# B&R Automation Studio project NAEUL004C00R13L518F00 (part 39)

#### Act_Main.st - Do Not Change!!!
```iecst
(** 2019-07-03 **)
ACTION Act_Main:

	fbMagPresentTm(IN := tylocalBuffer.In.bMagPresentSensor);

	//Update Retain
	IF bUpdateSensor = TRUE THEN
		tylocalBuffer.Out.bMagPresent	:= fbMagPresentTm.Q;
	END_IF

	//Display Buffer
	IF bUpdtDisplay = TRUE THEN
		fDispBffrDescending(ADR(tylocalBuffer.In.tyDispBuffer) , tyBffrParameter , tylocalBuffer.In.tyBuffer , tylocalBuffer.In.dtCurrDT , DINT_TO_TIME(tylocalBuffer.In.diCoolTm) , 0 , 1 , 2);
	END_IF

	//Cooling Fan Control
	IF tylocalBuffer.In.bManual = TRUE THEN
		;

	ELSIF bCoolFanRun = TRUE AND tylocalBuffer.In.bPrepCoolFan = TRUE AND bCoolFanTm = TRUE THEN //Cooling Fan Control By Cooling Time

		fbCoolFanOffChkTm(IN := TRUE);

		IF fbCoolFanOffChkTm.Q = TRUE THEN
			IF fBffrChkCoolBrdAny(tylocalBuffer.In.dtCurrDT, DINT_TO_TIME(tylocalBuffer.In.diCoolTm), tylocalBuffer.In.tyBuffer) = 0 THEN
				fbCoolFanOffDlyTm.IN	:= TRUE;
			ELSE
				fbCoolFanOffDlyTm.IN	:= FALSE;
				tylocalBuffer.Out.bCoolFanCtrl			:= TRUE;
			END_IF

			fbCoolFanOffChkTm(IN := FALSE);
		END_IF

		fbCoolFanOffDlyTm;

		IF fbCoolFanOffDlyTm.Q = TRUE THEN
			tylocalBuffer.Out.bCoolFanCtrl	:= FALSE;
		END_IF

	ELSIF bCoolFanRun = TRUE AND tylocalBuffer.In.bPrepCoolFan = TRUE AND bCoolFanTm = FALSE THEN	//Cooling Fan Control By Buffer Empty
		fbCoolFanOffDlyTm(IN := tylocalBuffer.In.tyBufferStat.bBffrMty);

		IF tylocalBuffer.In.tyBufferStat.bBffrMty = FALSE THEN
			tylocalBuffer.Out.bCoolFanCtrl	:= TRUE;
		END_IF

		IF fbCoolFanOffDlyTm.Q = TRUE THEN
			tylocalBuffer.Out.bCoolFanCtrl	:= FALSE;
		END_IF

	ELSE

		tylocalBuffer.Out.bCoolFanCtrl	:= FALSE;

	END_IF

	//Set Buffer By Magazine Present
	IF bBffrSetFull = TRUE THEN
		IF tylocalBuffer.In.bMagPresentSensor = TRUE AND fbMagAbsentTm.Q = TRUE THEN
			bSetFull		:= TRUE;
			tylocalBuffer.Out.dtMagPresentTm	:= tylocalBuffer.In.dtCurrDT;
		END_IF

		IF bSetFull = TRUE  THEN
			tylocalBuffer.In.eAct	:= BufferActSetFull;

			IF eStatus = Done AND eStat = BufferActSetFull THEN
				tylocalBuffer.In.eAct		:= BufferActIdle;
				bSetFull	:= FALSE;
			ELSIF eStatus = Error THEN
				bSetFull	:= FALSE;
			END_IF
		END_IF

		fbMagAbsentTm(IN := NOT tylocalBuffer.In.bMagPresentSensor);

	ELSIF bBffrSetMty = TRUE THEN
		IF tylocalBuffer.In.bMagPresentSensor = TRUE AND fbMagAbsentTm.Q = TRUE THEN
			bSetMty			:= TRUE;
			tylocalBuffer.Out.dtMagPresentTm	:= tylocalBuffer.In.dtCurrDT;
		END_IF

		IF bSetMty = TRUE  THEN
			tylocalBuffer.In.eAct	:= BufferActSetMty;

			IF eStatus = Done AND eStat = BufferActSetMty THEN
				tylocalBuffer.In.eAct	:= BufferActIdle;
				bSetMty	:= FALSE;
			ELSIF eStatus = Error THEN
				bSetMty	:= FALSE;
			END_IF
		END_IF

		fbMagAbsentTm(IN := NOT tylocalBuffer.In.bMagPresentSensor);

	END_IF
	//background--end//

	//Check Parameter Different
	tylocalBuffer.Out.bParamDiff	:= (tyBffrParameter.bAscending <> tylocalBuffer.In.bAscending)
	OR (tyBffrParameter.diMinSlt <> tylocalBuffer.In.diMinSlt)
	OR (tyBffrParameter.diMaxSlt <> tylocalBuffer.In.diMaxSlt)
	OR (tyBffrParameter.diPitch <> tylocalBuffer.In.diPitch)
	OR (tyBffrParameter.diSltCap <> tylocalBuffer.In.diSltCap)
	OR (tylocalBuffer.Out.bFIFOOld <> tylocalBuffer.In.bFIFO);

	//Update MagRemoved
	tylocalBuffer.Out.bMagRemoved	:= fbMagAbsentTm.Q;

	//Action
	IF tylocalBuffer.Out.eStatus = Idle OR tylocalBuffer.Out.eStatus = Busy OR tylocalBuffer.Out.eStatus = Done THEN
		tylocalBuffer.Out.eStat	:= tylocalBuffer.In.eAct;
	END_IF

	IF eStatOld <> tylocalBuffer.Out.eStat THEN
		fbDirCreate1(bEn := FALSE);
		fbDirCreate2(bEn := FALSE);
		fbFileRead1(bEn := FALSE);
		fbFileWrite1(bEn := FALSE);
		usiStep	:= 0;

		bFileNotFound			:= FALSE;
		bNewProduct				:= FALSE;
		bLastProductUnload		:= FALSE;
		bLastProductLeftInBffr	:= FALSE;

		tylocalBuffer.Out.sStatTxt	:= a_sStatText[tylocalBuffer.Out.eStat];

		eStatOld	:= tylocalBuffer.Out.eStat;

		tylocalBuffer.Out.eStatus		:= Busy;
	END_IF

	//Main
	CASE tylocalBuffer.Out.eStat OF

		BufferActIdle:
			tylocalBuffer.Out.eStatus	:= Idle;

		BufferActCreateDir:
			IF tylocalBuffer.Out.eStatus = Idle OR tylocalBuffer.Out.eStatus = Busy THEN

				tylocalBuffer.Out.eStatus	:= Busy;

				CASE usiStep OF
					0:
						fbDirCreate1(bEn := TRUE);
						IF fbDirCreate1.udiStatus = 0 THEN
							usiStep	:= 1;
						ELSIF fbDirCreate1.udiStatus < 65534 THEN
							tylocalBuffer.Out.eStatus		:= Error;

							IF fbDirCreate1.udiStatus = 1908 THEN
								udiStatus	:= 10000;	//Create User Directory Error
							ELSE
								udiStatus	:= fbDirCreate1.udiStatus;
							END_IF
						END_IF

					1:
						fbDirCreate2(bEn := TRUE);
						IF fbDirCreate2.udiStatus = 0 THEN
							tylocalBuffer.Out.eStatus	:= Done;
						ELSIF fbDirCreate2.udiStatus < 65534 THEN
							tylocalBuffer.Out.eStatus		:= Error;

							IF fbDirCreate2.udiStatus = 1908 THEN
								udiStatus	:= 10001;	//Create Retain Directory Error
							ELSE
								udiStatus	:= fbDirCreate2.udiStatus;
							END_IF
						END_IF

				END_CASE

			END_IF

		BufferActGetRetainBffr:
			IF tylocalBuffer.Out.eStatus = Idle OR tylocalBuffer.Out.eStatus = Busy THEN

				tylocalBuffer.Out.eStatus	:= Busy;

				fbFileRead1(bEn := TRUE);
				IF fbFileRead1.udiStatus = 0 THEN
					tylocalBuffer.Out.eStatus	:= Done;

					tyBffrParameter.diBffrTtlSlt	:= tylocalBuffer.In.diBffrTtlSlt;
					tyBffrParameter.diSltCap		:= tylocalBuffer.In.diSltCap;

					fBffrStat(ADR(tylocalBuffer.In.tylocalBuffer.Out.tylocalBuffer.Out.tyBufferStat) , tylocalBuffer.In.tylocalBuffer.Out.tyBuffer);
					fDispBffrDescending(ADR(tylocalBuffer.In.tylocalBuffer.Out.tyDispBuffer) , tyBffrParameter , tylocalBuffer.In.tylocalBuffer.Out.tyBuffer , tylocalBuffer.In.dtCurrDT , DINT_TO_TIME(tylocalBuffer.In.diCoolTm) , 0 , 1 , 2);

				ELSIF fbFileRead1.udiStatus < 65534 THEN
					tylocalBuffer.Out.eStatus	:= Error;

					IF fbFileRead1.udiStatus = 1900 THEN
						udiStatus	:= 10002;	//File Open Error While Reading Retain File
					ELSIF fbFileRead1.udiStatus = 1902 THEN
						udiStatus	:= 10003;	//File Read Error While Reading Retain File
					ELSIF fbFileRead1.udiStatus = 1904 THEN
						udiStatus	:= 10004;	//File Close Error While Reading Retain File
					ELSIF fbFileRead1.udiStatus = 1915 THEN
						tylocalBuffer.Out.eStatus			:= Done;
						bFileNotFound	:= TRUE;
					ELSE
						udiStatus	:= fbFileRead1.udiStatus;
					END_IF
				END_IF

			END_IF

		BufferActSetFull:
			IF tylocalBuffer.Out.eStatus = Idle OR tylocalBuffer.Out.eStatus = Busy THEN

				tylocalBuffer.Out.eStatus	:= Busy;

				CASE usiStep OF
					0:
						tyBffrParameter.bAscending		:= tylocalBuffer.In.bAscending;
						tyBffrParameter.diBffrTtlSlt	:= tylocalBuffer.In.diBffrTtlSlt;
						tyBffrParameter.diMaxSlt		:= tylocalBuffer.In.diMaxSlt;
						tyBffrParameter.diMinSlt		:= tylocalBuffer.In.diMinSlt;
						tyBffrParameter.diPitch			:= tylocalBuffer.In.diPitch;
						tyBffrParameter.diSltCap		:= tylocalBuffer.In.diSltCap;
						tyBffrParameter.a_bSkip			:= tylocalBuffer.In.a_bSkip;
						tylocalBuffer.Out.bFIFOOld		:= tylocalBuffer.In.bFIFO;

						udiStatus	:= fBffrSetFull(ADR(tylocalBuffer.In.tylocalBuffer.Out.tyBuffer) , tyBffrParameter , tylocalBuffer.In.dtCurrDT , tylocalBuffer.In.sBffrNm , tylocalBuffer.In.sProdNm);

						IF udiStatus = 0 THEN
							usiStep	:= 1;

							fBffrStat(ADR(tylocalBuffer.In.tylocalBuffer.Out.tylocalBuffer.Out.tyBufferStat) , tylocalBuffer.In.tylocalBuffer.Out.tyBuffer);
							fDispBffrDescending(ADR(tylocalBuffer.In.tylocalBuffer.Out.tyDispBuffer) , tyBffrParameter , tylocalBuffer.In.tylocalBuffer.Out.tyBuffer , tylocalBuffer.In.dtCurrDT , DINT_TO_TIME(tylocalBuffer.In.diCoolTm) , 0 , 1 , 2);

						ELSE
							tylocalBuffer.Out.eStatus	:= Error;

						END_IF

					1:
						fbFileWrite1(bEn := TRUE);

						IF fbFileWrite1.udiStatus = 0 THEN
							tylocalBuffer.Out.eStatus	:= Done;
						ELSIF fbFileWrite1.udiStatus < 65534 THEN
							tylocalBuffer.Out.eStatus	:= Error;

							IF fbFileWrite1.udiStatus = 1900 THEN
								udiStatus	:= 10005;	//File Open Error While Setting Full Buffer
							ELSIF fbFileWrite1.udiStatus = 1901 THEN
								udiStatus	:= 10006;	//File Create Error While Setting Full Buffer
							ELSIF fbFileWrite1.udiStatus = 1903 THEN
								udiStatus	:= 10007;	//File Write Error While Setting Full Buffer
							ELSIF fbFileWrite1.udiStatus = 1904 THEN
								udiStatus	:= 10008;	//File Close Error While Setting Full Buffer
							ELSIF fbFileWrite1.udiStatus = 1914 THEN
								udiStatus	:= 10040;	//Directory Does Not Exist While Setting Full Buffer
							ELSE
								udiStatus	:= fbFileWrite1.udiStatus;
							END_IF
						END_IF

				END_CASE

			END_IF

		BufferActSetMty:
			IF tylocalBuffer.Out.eStatus = Idle OR tylocalBuffer.Out.eStatus = Busy THEN

				tylocalBuffer.Out.eStatus	:= Busy;

				CASE usiStep OF
					0:
						tyBffrParameter.bAscending		:= tylocalBuffer.In.bAscending;
						tyBffrParameter.diBffrTtlSlt	:= tylocalBuffer.In.diBffrTtlSlt;
						tyBffrParameter.diMaxSlt		:= tylocalBuffer.In.diMaxSlt;
						tyBffrParameter.diMinSlt		:= tylocalBuffer.In.diMinSlt;
						tyBffrParameter.diPitch			:= tylocalBuffer.In.diPitch;
						tyBffrParameter.diSltCap		:= tylocalBuffer.In.diSltCap;
						tyBffrParameter.a_bSkip			:= tylocalBuffer.In.a_bSkip;
						tylocalBuffer.Out.bFIFOOld						:= tylocalBuffer.In.bFIFO;

						udiStatus	:= fBffrSetMty(ADR(tylocalBuffer.In.tylocalBuffer.Out.tyBuffer) , tyBffrParameter , tylocalBuffer.In.sBffrNm);

						IF udiStatus = 0 THEN
							usiStep	:= 1;

							fBffrStat(ADR(tylocalBuffer.In.tylocalBuffer.Out.tylocalBuffer.Out.tyBufferStat) , tylocalBuffer.In.tylocalBuffer.Out.tyBuffer);
							fDispBffrDescending(ADR(tylocalBuffer.In.tylocalBuffer.Out.tyDispBuffer) , tyBffrParameter , tylocalBuffer.In.tylocalBuffer.Out.tyBuffer , tylocalBuffer.In.dtCurrDT , DINT_TO_TIME(tylocalBuffer.In.diCoolTm) , 0 , 1 , 2);

						ELSE
							tylocalBuffer.Out.eStatus	:= Error;

						END_IF

					1:
						fbFileWrite1(bEn := TRUE);

						IF fbFileWrite1.udiStatus = 0 THEN
							tylocalBuffer.Out.eStatus	:= Done;
						ELSIF fbFileWrite1.udiStatus < 65534 THEN
							tylocalBuffer.Out.eStatus	:= Error;

							IF fbFileWrite1.udiStatus = 1900 THEN
								udiStatus	:= 10009;	//File Open Error While Setting Empty Buffer
							ELSIF fbFileWrite1.udiStatus = 1901 THEN
								udiStatus	:= 10010;	//File Create Error While Setting Empty Buffer
							ELSIF fbFileWrite1.udiStatus = 1903 THEN
								udiStatus	:= 10011;	//File Write Error While Setting Empty Buffer
							ELSIF fbFileWrite1.udiStatus = 1904 THEN
								udiStatus	:= 10012;	//File Close Error While Setting Empty Buffer
							ELSIF fbFileWrite1.udiStatus = 1914 THEN
								udiStatus	:= 10041;	//Directory Does Not Exist While Setting Empty Buffer
							ELSE
								udiStatus	:= fbFileWrite1.udiStatus;
							END_IF
						END_IF

				END_CASE

			END_IF

		BufferActLoad:
			IF tylocalBuffer.Out.eStatus = Idle OR tylocalBuffer.Out.eStatus = Busy THEN

				tylocalBuffer.Out.eStatus	:= Busy;

				CASE usiStep OF
					0:
						tyLocalBuffer.Out.diCurrSlt	:= fLifterPosInUMToSltBtmMin(tylocalBuffer.In.diLifterCurrPosInUM , tylocalBuffer.In.diSltToSltInUM , tylocalBuffer.In.diLifterBtmPosInUM);

						udiStatus	:= fBffrLoad(ADR(tylocalBuffer.In.tylocalBuffer.Out.tyBuffer) , ADR(bNewProduct) , tyLocalBuffer.Out.diCurrSlt , tylocalBuffer.In.dtCurrDT , tylocalBuffer.In.bGdBrdIn , tylocalBuffer.In.sProdNm , tylocalBuffer.In.sBarcode1 , tylocalBuffer.In.sBarcode2);

						IF udiStatus = 0 THEN
							usiStep	:= 1;

							tyBffrParameter.diBffrTtlSlt	:= tylocalBuffer.In.diBffrTtlSlt;
							tyBffrParameter.diSltCap		:= tylocalBuffer.In.diSltCap;

							fBffrStat(ADR(tylocalBuffer.In.tylocalBuffer.Out.tylocalBuffer.Out.tyBufferStat) , tylocalBuffer.In.tylocalBuffer.Out.tyBuffer);
							fDispBffrDescending(ADR(tylocalBuffer.In.tylocalBuffer.Out.tyDispBuffer) , tyBffrParameter , tylocalBuffer.In.tylocalBuffer.Out.tyBuffer , tylocalBuffer.In.dtCurrDT , DINT_TO_TIME(tylocalBuffer.In.diCoolTm) , 0 , 1 , 2);

						ELSE
							tylocalBuffer.Out.eStatus	:= Error;

							IF udiStatus = 1010 THEN
								udiStatus	:= 10076;	//Loading Slot Is Not For Board
							ELSIF udiStatus = 1011 THEN
								udiStatus	:= 10077;	//Loading Slot Is Full Of Board
							ELSIF udiStatus = 1012 THEN
								udiStatus	:= 10078;	//Loading First Sub-Slot Is Not For Board
							ELSIF udiStatus	= 1013 THEN
								udiStatus	:= 10079;	//Loading Last Sub-Slot Have Board, Which Mean Slot Is Full Of Board
							ELSIF udiStatus = 1014 THEN
								udiStatus	:= 10080;	//Loading Last Sub-Slot Is Not For Board
							ELSIF udiStatus = 1015 THEN
								udiStatus	:= 10081;	//Loading Slot Is Full Of Board
							ELSIF udiStatus = 1001 THEN
								udiStatus	:= 10082;	//Loading Slot Is Skipped
							ELSIF udiStatus	= 1016 THEN
								udiStatus	:= 10083;	//Existing Board Status Is Different With Loading Board Status
							END_IF

						END_IF

					1:
						fbFileWrite1(bEn := TRUE);

						IF fbFileWrite1.udiStatus = 0 THEN
							tylocalBuffer.Out.eStatus	:= Done;
						ELSIF fbFileWrite1.udiStatus < 65534 THEN
							tylocalBuffer.Out.eStatus	:= Error;

							IF fbFileWrite1.udiStatus = 1900 THEN
								udiStatus	:= 10013;	//File Open Error While Loading Info To Buffer
							ELSIF fbFileWrite1.udiStatus = 1901 THEN
								udiStatus	:= 10014;	//File Create Error While Loading Info To Buffer
							ELSIF fbFileWrite1.udiStatus = 1903 THEN
								udiStatus	:= 10015;	//File Write Error While Loading Info To Buffer
							ELSIF fbFileWrite1.udiStatus = 1904 THEN
								udiStatus	:= 10016;	//File Close Error While Loading Info To Buffer
							ELSIF fbFileWrite1.udiStatus = 1914 THEN
								udiStatus	:= 10042;	//Directory Does Not Exist While Loading Info To Buffer
							ELSE
								udiStatus	:= fbFileWrite1.udiStatus;
							END_IF
						END_IF

				END_CASE

			END_IF

		BufferActLoadSltChk:
			IF tylocalBuffer.Out.eStatus = Idle OR tylocalBuffer.Out.eStatus = Busy THEN

				tylocalBuffer.Out.eStatus	:= Busy;

				CASE usiStep OF
					0:
						tyLocalBuffer.Out.diCurrSlt	:= fLifterPosInUMToSltBtmMin(tylocalBuffer.In.diLifterCurrPosInUM , tylocalBuffer.In.diSltToSltInUM , tylocalBuffer.In.diLifterBtmPosInUM);

						IF tylocalBuffer.In.bNxtLoadSeq = TRUE AND tylocalBuffer.In.bGdBrdIn = TRUE THEN
							diExpectedSlt	:= fBffrNxtLoadSeqGd(tylocalBuffer.In.bAscending , tylocalBuffer.In.tylocalBuffer.Out.tyBuffer);
						ELSIF tylocalBuffer.In.bNxtLoadSeq = TRUE AND tylocalBuffer.In.bGdBrdIn = FALSE THEN
							diExpectedSlt	:= fBffrNxtLoadSeqBad(tylocalBuffer.In.bAscending , tylocalBuffer.In.tylocalBuffer.Out.tyBuffer);
						ELSIF tylocalBuffer.In.bNxtLoadSeq = FALSE AND tylocalBuffer.In.bGdBrdIn = TRUE THEN
							diExpectedSlt	:= fBffrNxtLoadNearbyGd(tyLocalBuffer.Out.diCurrSlt , tylocalBuffer.In.tylocalBuffer.Out.tyBuffer);
						ELSE
							diExpectedSlt	:= fBffrNxtLoadNearbyBad(tyLocalBuffer.Out.diCurrSlt , tylocalBuffer.In.tylocalBuffer.Out.tyBuffer);
						END_IF

						IF tyLocalBuffer.Out.diCurrSlt = diExpectedSlt THEN
							udiStatus	:= fBffrLoad(ADR(tylocalBuffer.In.tylocalBuffer.Out.tyBuffer) , ADR(bNewProduct) , tyLocalBuffer.Out.diCurrSlt , tylocalBuffer.In.dtCurrDT , tylocalBuffer.In.bGdBrdIn , tylocalBuffer.In.sProdNm , tylocalBuffer.In.sBarcode1 , tylocalBuffer.In.sBarcode2);

							IF udiStatus = 0 THEN
								usiStep	:= 1;

								tyBffrParameter.diBffrTtlSlt	:= tylocalBuffer.In.diBffrTtlSlt;
								tyBffrParameter.diSltCap		:= tylocalBuffer.In.diSltCap;

								fBffrStat(ADR(tylocalBuffer.In.tylocalBuffer.Out.tylocalBuffer.Out.tyBufferStat) , tylocalBuffer.In.tylocalBuffer.Out.tyBuffer);
								fDispBffrDescending(ADR(tylocalBuffer.In.tylocalBuffer.Out.tyDispBuffer) , tyBffrParameter , tylocalBuffer.In.tylocalBuffer.Out.tyBuffer , tylocalBuffer.In.dtCurrDT , DINT_TO_TIME(tylocalBuffer.In.diCoolTm) , 0 , 1 , 2);

							ELSE
								tylocalBuffer.Out.eStatus	:= Error;

								IF udiStatus = 1010 THEN
									udiStatus	:= 10084;	//Loading Slot Is Not For Board
								ELSIF udiStatus = 1011 THEN
									udiStatus	:= 10085;	//Loading Slot Is Full Of Board
								ELSIF udiStatus = 1012 THEN
									udiStatus	:= 10086;	//Loading First Sub-Slot Is Not For Board
								ELSIF udiStatus	= 1013 THEN
									udiStatus	:= 10087;	//Loading Last Sub-Slot Have Board, Which Mean Slot Is Full Of Board
								ELSIF udiStatus = 1014 THEN
									udiStatus	:= 10088;	//Loading Last Sub-Slot Is Not For Board
								ELSIF udiStatus = 1015 THEN
									udiStatus	:= 10089;	//Loading Slot Is Full Of Board
								ELSIF udiStatus = 1001 THEN
									udiStatus	:= 10090;	//Loading Slot Is Skipped
								ELSIF udiStatus	= 1016 THEN
									udiStatus	:= 10091;	//Existing Board Status Is Different With Loading Board Status
								END_IF

							END_IF

						ELSE
							udiStatus	:= 10017;	//Wrong Slot Number To Load
							tylocalBuffer.Out.eStatus		:= Error;

						END_IF

					1:
						fbFileWrite1(bEn := TRUE);

						IF fbFileWrite1.udiStatus = 0 THEN
							tylocalBuffer.Out.eStatus	:= Done;
						ELSIF fbFileWrite1.udiStatus < 65534 THEN
							tylocalBuffer.Out.eStatus	:= Error;

							IF fbFileWrite1.udiStatus = 1900 THEN
								udiStatus	:= 10018;	//File Open Error While Loading Info To Buffer With Slot Check
							ELSIF fbFileWrite1.udiStatus = 1901 THEN
								udiStatus	:= 10019;	//File Create Error While Loading Info To Buffer With Slot Check
							ELSIF fbFileWrite1.udiStatus = 1903 THEN
								udiStatus	:= 10020;	//File Write Error While Loading Info To Buffer With Slot Check
							ELSIF fbFileWrite1.udiStatus = 1904 THEN
								udiStatus	:= 10021;	//File Close Error While Loading Info To Buffer With Slot Check
							ELSIF fbFileWrite1.udiStatus = 1914 THEN
								udiStatus	:= 10043;	//Directory Does Not Exist While Loading Info To Buffer With Slot Check
							ELSE
								udiStatus	:= fbFileWrite1.udiStatus;
							END_IF
						END_IF

				END_CASE

			END_IF

		BufferActUnload:
			IF tylocalBuffer.Out.eStatus = Idle OR tylocalBuffer.Out.eStatus = Busy THEN

				tylocalBuffer.Out.eStatus	:= Busy;

				CASE usiStep OF
					0:
						tyLocalBuffer.Out.diCurrSlt	:= fLifterPosInUMToSltBtmMin(tylocalBuffer.In.diLifterCurrPosInUM , tylocalBuffer.In.diSltToSltInUM , tylocalBuffer.In.diLifterBtmPosInUM);

						udiStatus	:= fBffrUnload(ADR(tylocalBuffer.Out.tyBoardUnloadStat) , ADR(tylocalBuffer.In.tylocalBuffer.Out.tyBuffer) , ADR(bLastProductUnload) , ADR(bLastProductLeftInBffr) , tyLocalBuffer.Out.diCurrSlt);

						IF tylocalBuffer.In.sCurrRcpNm = tylocalBuffer.Out.tyBoardUnloadStat.sProdNm THEN
							bLastProductUnload	:= FALSE;
						END_IF

						IF udiStatus = 0 THEN
							usiStep	:= 1;

							tyBffrParameter.diBffrTtlSlt	:= tylocalBuffer.In.diBffrTtlSlt;
							tyBffrParameter.diSltCap		:= tylocalBuffer.In.diSltCap;

							fBffrStat(ADR(tylocalBuffer.In.tylocalBuffer.Out.tylocalBuffer.Out.tyBufferStat) , tylocalBuffer.In.tylocalBuffer.Out.tyBuffer);
							fDispBffrDescending(ADR(tylocalBuffer.In.tylocalBuffer.Out.tyDispBuffer) , tyBffrParameter , tylocalBuffer.In.tylocalBuffer.Out.tyBuffer , tylocalBuffer.In.dtCurrDT , DINT_TO_TIME(tylocalBuffer.In.diCoolTm) , 0 , 1 , 2);

						ELSE
							tylocalBuffer.Out.eStatus	:= Error;

							IF udiStatus = 1000 THEN
								udiStatus	:= 10048;	//Unloading Slot Is Skipped While Unloading Buffer
							ELSIF udiStatus = 1003 THEN
								udiStatus	:= 10049;	//Unloading Slot Is Not For Board While Unloading Buffer
							ELSIF udiStatus = 1004 THEN
								udiStatus	:= 10050;	//Unloading Slot Board Is Not available While Unloading Buffer
							ELSIF udiStatus = 1005 THEN
								udiStatus	:= 10051;	//Unloading Last Sub Slot Is Not For Board While Unloading Buffer
							ELSIF udiStatus = 1006 THEN
								udiStatus	:= 10052;	//Unloading Last Sub Slot Has No Board While Unloading Buffer
							ELSIF udiStatus = 1007 THEN
								udiStatus	:= 10053;	//Board Quantity In Slot Is 0 While Unloading Buffer
							ELSIF udiStatus = 1008 THEN
								udiStatus	:= 10054;	//Board Capacity In Slot Is 0 While Unloading Buffer
							END_IF

						END_IF

					1:
						fbFileWrite1(bEn := TRUE);

						IF fbFileWrite1.udiStatus = 0 THEN
							tylocalBuffer.Out.eStatus	:= Done;
						ELSIF fbFileWrite1.udiStatus < 65534 THEN
							tylocalBuffer.Out.eStatus	:= Error;

							IF fbFileWrite1.udiStatus = 1900 THEN
								udiStatus	:= 10022;	//File Open Error While Unloading Info From Buffer
							ELSIF fbFileWrite1.udiStatus = 1901 THEN
								udiStatus	:= 10023;	//File Create Error While Unloading Info From Buffer
							ELSIF fbFileWrite1.udiStatus = 1903 THEN
								udiStatus	:= 10024;	//File Write Error While Unloading Info From Buffer
							ELSIF fbFileWrite1.udiStatus = 1904 THEN
								udiStatus	:= 10025;	//File Close Error While Unloading Info From Buffer
							ELSIF fbFileWrite1.udiStatus = 1914 THEN
								udiStatus	:= 10044;	//Directory Does Not Exist While Unloading Info From Buffer
							ELSE
								udiStatus	:= fbFileWrite1.udiStatus;
							END_IF
						END_IF

				END_CASE

			END_IF

		BufferActUnloadSltChk:
			IF tylocalBuffer.Out.eStatus = Idle OR tylocalBuffer.Out.eStatus = Busy THEN

				tylocalBuffer.Out.eStatus	:= Busy;

				CASE usiStep OF
					0:
						tyLocalBuffer.Out.diCurrSlt	:= fLifterPosInUMToSltBtmMin(tylocalBuffer.In.diLifterCurrPosInUM , tylocalBuffer.In.diSltToSltInUM , tylocalBuffer.In.diLifterBtmPosInUM);

						IF tylocalBuffer.In.bFIFO = TRUE AND tylocalBuffer.In.bGdBrdReq = TRUE THEN
							diExpectedSlt	:= fBffrNxtUnloadFIFOGd(tylocalBuffer.In.tylocalBuffer.Out.tyBuffer , '');
						ELSIF tylocalBuffer.In.bFIFO = TRUE AND tylocalBuffer.In.bGdBrdReq = FALSE THEN
							diExpectedSlt	:= fBffrNxtUnloadFIFOBad(tylocalBuffer.In.tylocalBuffer.Out.tyBuffer , '');
						ELSIF tylocalBuffer.In.bFIFO = FALSE AND tylocalBuffer.In.bGdBrdReq = TRUE THEN
							diExpectedSlt	:= fBffrNxtUnloadLIFOGd(tylocalBuffer.In.tylocalBuffer.Out.tyBuffer , '');
						ELSE
							diExpectedSlt	:= fBffrNxtUnloadLIFOBad(tylocalBuffer.In.tylocalBuffer.Out.tyBuffer , '');
						END_IF

						IF tyLocalBuffer.Out.diCurrSlt = diExpectedSlt THEN
							udiStatus	:= fBffrUnload(ADR(tylocalBuffer.Out.tyBoardUnloadStat) , ADR(tylocalBuffer.In.tylocalBuffer.Out.tyBuffer) , ADR(bLastProductUnload) , ADR(bLastProductLeftInBffr) , tyLocalBuffer.Out.diCurrSlt);

							IF tylocalBuffer.In.sCurrRcpNm = tylocalBuffer.Out.tyBoardUnloadStat.sProdNm THEN
								bLastProductUnload	:= FALSE;
							END_IF

							IF udiStatus = 0 THEN
								usiStep	:= 1;

								tyBffrParameter.diBffrTtlSlt	:= tylocalBuffer.In.diBffrTtlSlt;
								tyBffrParameter.diSltCap		:= tylocalBuffer.In.diSltCap;

								fBffrStat(ADR(tylocalBuffer.In.tylocalBuffer.Out.tylocalBuffer.Out.tyBufferStat) , tylocalBuffer.In.tylocalBuffer.Out.tyBuffer);
								fDispBffrDescending(ADR(tylocalBuffer.In.tylocalBuffer.Out.tyDispBuffer) , tyBffrParameter , tylocalBuffer.In.tylocalBuffer.Out.tyBuffer , tylocalBuffer.In.dtCurrDT , DINT_TO_TIME(tylocalBuffer.In.diCoolTm) , 0 , 1 , 2);

							ELSE
								tylocalBuffer.Out.eStatus	:= Error;

								IF udiStatus = 1000 THEN
									udiStatus	:= 10055;	//Unloading Slot Is Skipped While Unloading Buffer With Slot Check
								ELSIF udiStatus = 1003 THEN
									udiStatus	:= 10056;	//Unloading Slot Is Not For Board While Unloading Buffer With Slot Check
								ELSIF udiStatus = 1004 THEN
									udiStatus	:= 10057;	//Unloading Slot Board Is Not available While Unloading Buffer With Slot Check
								ELSIF udiStatus = 1005 THEN
									udiStatus	:= 10058;	//Unloading Last Sub Slot Is Not For Board While Unloading Buffer With Slot Check
								ELSIF udiStatus = 1006 THEN
									udiStatus	:= 10059;	//Unloading Last Sub Slot Has No Board While Unloading Buffer With Slot Check
								ELSIF udiStatus = 1007 THEN
									udiStatus	:= 10060;	//Board Quantity In Slot Is 0 While Unloading Buffer With Slot Check
								ELSIF udiStatus = 1008 THEN
									udiStatus	:= 10061;	//Board Capacity In Slot Is 0 While Unloading Buffer With Slot Check
								END_IF

							END_IF

						ELSE
							udiStatus	:= 10026;	//Wrong Slot Number To Unload
							tylocalBuffer.Out.eStatus		:= Error;

						END_IF

					1:
						fbFileWrite1(bEn := TRUE);

						IF fbFileWrite1.udiStatus = 0 THEN
							tylocalBuffer.Out.eStatus	:= Done;
						ELSIF fbFileWrite1.udiStatus < 65534 THEN
							tylocalBuffer.Out.eStatus	:= Error;

							IF fbFileWrite1.udiStatus = 1900 THEN
								udiStatus	:= 10027;	//File Open Error While Unloading Info From Buffer With Slot Check
							ELSIF fbFileWrite1.udiStatus = 1901 THEN
								udiStatus	:= 10028;	//File Create Error While Unloading Info From Buffer With Slot Check
							ELSIF fbFileWrite1.udiStatus = 1903 THEN
								udiStatus	:= 10029;	//File Write Error While Unloading Info From Buffer With Slot Check
							ELSIF fbFileWrite1.udiStatus = 1904 THEN
								udiStatus	:= 10030;	//File Close Error While Unloading Info From Buffer With Slot Check
							ELSIF fbFileWrite1.udiStatus = 1914 THEN
								udiStatus	:= 10045;	//Directory Does Not Exist While Unloading Info From Buffer With Slot Check
							ELSE
								udiStatus	:= fbFileWrite1.udiStatus;
							END_IF
						END_IF

				END_CASE

			END_IF

		BufferActUnloadCoolChk:
			IF tylocalBuffer.Out.eStatus = Idle OR tylocalBuffer.Out.eStatus = Busy THEN

				tylocalBuffer.Out.eStatus	:= Busy;

				CASE usiStep OF
					0:
						tyLocalBuffer.Out.diCurrSlt	:= fLifterPosInUMToSltBtmMin(tylocalBuffer.In.diLifterCurrPosInUM , tylocalBuffer.In.diSltToSltInUM , tylocalBuffer.In.diLifterBtmPosInUM);

						tylocalBuffer.Out.bCoolNotRdy	:= NOT fBffrChkCoolTmRdy(tyLocalBuffer.Out.diCurrSlt, tylocalBuffer.In.dtCurrDT, DINT_TO_TIME(tylocalBuffer.In.diCoolTm), tylocalBuffer.In.tylocalBuffer.Out.tyBuffer);

						IF tylocalBuffer.Out.bCoolNotRdy = FALSE THEN
							udiStatus	:= fBffrUnload(ADR(tylocalBuffer.Out.tyBoardUnloadStat) , ADR(tylocalBuffer.In.tylocalBuffer.Out.tyBuffer) , ADR(bLastProductUnload) , ADR(bLastProductLeftInBffr) , tyLocalBuffer.Out.diCurrSlt);

							IF tylocalBuffer.In.sCurrRcpNm = tylocalBuffer.Out.tyBoardUnloadStat.sProdNm THEN
								bLastProductUnload	:= FALSE;
							END_IF

							IF udiStatus = 0 THEN
								usiStep	:= 1;

								tyBffrParameter.diBffrTtlSlt	:= tylocalBuffer.In.diBffrTtlSlt;
								tyBffrParameter.diSltCap		:= tylocalBuffer.In.diSltCap;

								fBffrStat(ADR(tylocalBuffer.In.tylocalBuffer.Out.tylocalBuffer.Out.tyBufferStat) , tylocalBuffer.In.tylocalBuffer.Out.tyBuffer);
								fDispBffrDescending(ADR(tylocalBuffer.In.tylocalBuffer.Out.tyDispBuffer) , tyBffrParameter , tylocalBuffer.In.tylocalBuffer.Out.tyBuffer , tylocalBuffer.In.dtCurrDT , DINT_TO_TIME(tylocalBuffer.In.diCoolTm) , 0 , 1 , 2);

							ELSE
								tylocalBuffer.Out.eStatus	:= Error;

								IF udiStatus = 1000 THEN
									udiStatus	:= 10062;	//Unloading Slot Is Skipped While Unloading Buffer With Cool Check
								ELSIF udiStatus = 1003 THEN
									udiStatus	:= 10063;	//Unloading Slot Is Not For Board While Unloading Buffer With Cool Check
								ELSIF udiStatus = 1004 THEN
									udiStatus	:= 10064;	//Unloading Slot Board Is Not available While Unloading Buffer With Cool Check
								ELSIF udiStatus = 1005 THEN
									udiStatus	:= 10065;	//Unloading Last Sub Slot Is Not For Board While Unloading Buffer With Cool Check
								ELSIF udiStatus = 1006 THEN
									udiStatus	:= 10066;	//Unloading Last Sub Slot Has No Board While Unloading Buffer With Cool Check
								ELSIF udiStatus = 1007 THEN
									udiStatus	:= 10067;	//Board Quantity In Slot Is 0 While Unloading Buffer With Cool Check
								ELSIF udiStatus = 1008 THEN
									udiStatus	:= 10068;	//Board Capacity In Slot Is 0 While Unloading Buffer With Cool Check
								END_IF

							END_IF

						ELSE
							tylocalBuffer.Out.eStatus	:= Done;

						END_IF

					1:
						fbFileWrite1(bEn := TRUE);

						IF fbFileWrite1.udiStatus = 0 THEN
							tylocalBuffer.Out.eStatus	:= Done;
						ELSIF fbFileWrite1.udiStatus < 65534 THEN
							tylocalBuffer.Out.eStatus	:= Error;

							IF fbFileWrite1.udiStatus = 1900 THEN
								udiStatus	:= 10031;	//File Open Error While Unloading Info From Buffer With Cooling Time Check
							ELSIF fbFileWrite1.udiStatus = 1901 THEN
								udiStatus	:= 10032;	//File Create Error While Unloading Info From Buffer With Cooling Time Check
							ELSIF fbFileWrite1.udiStatus = 1903 THEN
								udiStatus	:= 10033;	//File Write Error While Unloading Info From Buffer With Cooling Time Check
							ELSIF fbFileWrite1.udiStatus = 1904 THEN
								udiStatus	:= 10034;	//File Close Error While Unloading Info From Buffer With Cooling Time Check
							ELSIF fbFileWrite1.udiStatus = 1914 THEN
								udiStatus	:= 10046;	//Directory Does Not Exist While Unloading Info From Buffer With Cooling Time Check
							ELSE
								udiStatus	:= fbFileWrite1.udiStatus;
							END_IF
						END_IF

				END_CASE

			END_IF

		BufferActUnloadSltChkCoolChk:
			IF tylocalBuffer.Out.eStatus = Idle OR tylocalBuffer.Out.eStatus = Busy THEN

				tylocalBuffer.Out.eStatus	:= Busy;

				CASE usiStep OF
					0:
						tyLocalBuffer.Out.diCurrSlt	:= fLifterPosInUMToSltBtmMin(tylocalBuffer.In.diLifterCurrPosInUM , tylocalBuffer.In.diSltToSltInUM , tylocalBuffer.In.diLifterBtmPosInUM);

						IF tylocalBuffer.In.bFIFO = TRUE AND tylocalBuffer.In.bGdBrdReq = TRUE THEN
							diExpectedSlt	:= fBffrNxtUnloadFIFOGd(tylocalBuffer.In.tylocalBuffer.Out.tyBuffer , '');
						ELSIF tylocalBuffer.In.bFIFO = TRUE AND tylocalBuffer.In.bGdBrdReq = FALSE THEN
							diExpectedSlt	:= fBffrNxtUnloadFIFOBad(tylocalBuffer.In.tylocalBuffer.Out.tyBuffer , '');
						ELSIF tylocalBuffer.In.bFIFO = FALSE AND tylocalBuffer.In.bGdBrdReq = TRUE THEN
							diExpectedSlt	:= fBffrNxtUnloadLIFOGd(tylocalBuffer.In.tylocalBuffer.Out.tyBuffer , '');
						ELSE
							diExpectedSlt	:= fBffrNxtUnloadLIFOBad(tylocalBuffer.In.tylocalBuffer.Out.tyBuffer , '');
						END_IF

						IF tyLocalBuffer.Out.diCurrSlt = diExpectedSlt THEN
							tylocalBuffer.Out.bCoolNotRdy	:= NOT fBffrChkCoolTmRdy(tyLocalBuffer.Out.diCurrSlt, tylocalBuffer.In.dtCurrDT, DINT_TO_TIME(tylocalBuffer.In.diCoolTm), tylocalBuffer.In.tylocalBuffer.Out.tyBuffer);

							IF tylocalBuffer.Out.bCoolNotRdy = FALSE THEN
								udiStatus	:= fBffrUnload(ADR(tylocalBuffer.Out.tyBoardUnloadStat) , ADR(tylocalBuffer.In.tylocalBuffer.Out.tyBuffer) , ADR(bLastProductUnload) , ADR(bLastProductLeftInBffr) , tyLocalBuffer.Out.diCurrSlt);

								IF tylocalBuffer.In.sCurrRcpNm = tylocalBuffer.Out.tyBoardUnloadStat.sProdNm THEN
									bLastProductUnload	:= FALSE;
								END_IF

								IF udiStatus = 0 THEN
									usiStep	:= 1;

									tyBffrParameter.diBffrTtlSlt	:= tylocalBuffer.In.diBffrTtlSlt;
									tyBffrParameter.diSltCap		:= tylocalBuffer.In.diSltCap;

									fBffrStat(ADR(tylocalBuffer.In.tylocalBuffer.Out.tylocalBuffer.Out.tyBufferStat) , tylocalBuffer.In.tylocalBuffer.Out.tyBuffer);
									fDispBffrDescending(ADR(tylocalBuffer.In.tylocalBuffer.Out.tyDispBuffer) , tyBffrParameter , tylocalBuffer.In.tylocalBuffer.Out.tyBuffer , tylocalBuffer.In.dtCurrDT , DINT_TO_TIME(tylocalBuffer.In.diCoolTm) , 0 , 1 , 2);

								ELSE
									tylocalBuffer.Out.eStatus	:= Error;

									IF udiStatus = 1000 THEN
										udiStatus	:= 10069;	//Unloading Slot Is Skipped While Unloading Buffer With Cool & Slot Check
									ELSIF udiStatus = 1003 THEN
										udiStatus	:= 10070;	//Unloading Slot Is Not For Board While Unloading Buffer With Cool & Slot Check
									ELSIF udiStatus = 1004 THEN
										udiStatus	:= 10071;	//Unloading Slot Board Is Not available While Unloading Buffer With Cool & Slot Check
									ELSIF udiStatus = 1005 THEN
										udiStatus	:= 10072;	//Unloading Last Sub Slot Is Not For Board While Unloading Buffer With Cool & Slot Check
									ELSIF udiStatus = 1006 THEN
										udiStatus	:= 10073;	//Unloading Last Sub Slot Has No Board While Unloading Buffer With Cool & Slot Check
									ELSIF udiStatus = 1007 THEN
										udiStatus	:= 10074;	//Board Quantity In Slot Is 0 While Unloading Buffer With Cool & Slot Check
									ELSIF udiStatus = 1008 THEN
										udiStatus	:= 10075;	//Board Capacity In Slot Is 0 While Unloading Buffer With Cool & Slot Check
									END_IF

								END_IF

							ELSE
								tylocalBuffer.Out.eStatus	:= Done;

							END_IF

						ELSE
							udiStatus	:= 10035;	//Wrong Slot Number To Unload With Cooling Time Check
							tylocalBuffer.Out.eStatus		:= Error;

						END_IF

					1:
						fbFileWrite1(bEn := TRUE);

						IF fbFileWrite1.udiStatus = 0 THEN
							tylocalBuffer.Out.eStatus	:= Done;
						ELSIF fbFileWrite1.udiStatus < 65534 THEN
							tylocalBuffer.Out.eStatus	:= Error;

							IF fbFileWrite1.udiStatus = 1900 THEN
								udiStatus	:= 10036;	//File Open Error While Unloading Info From Buffer With Slot Check And Cooling Time Check
							ELSIF fbFileWrite1.udiStatus = 1901 THEN
								udiStatus	:= 10037;	//File Create Error While Unloading Info From Buffer With Slot Check And Cooling Time Check
							ELSIF fbFileWrite1.udiStatus = 1903 THEN
								udiStatus	:= 10038;	//File Write Error While Unloading Info From Buffer With Slot Check And Cooling Time Check
							ELSIF fbFileWrite1.udiStatus = 1904 THEN
								udiStatus	:= 10039;	//File Close Error While Unloading Info From Buffer With Slot Check And Cooling Time Check
							ELSIF fbFileWrite1.udiStatus = 1914 THEN
								udiStatus	:= 10047;	//Directory Does Not Exist While Unloading Info From Buffer With Slot Check And Cooling Time Check
							ELSE
								udiStatus	:= fbFileWrite1.udiStatus;
							END_IF
						END_IF

				END_CASE

			END_IF

		BufferActNxtLoad:
			IF tylocalBuffer.Out.eStatus = Idle OR tylocalBuffer.Out.eStatus = Busy THEN

				tyLocalBuffer.Out.diCurrSlt	:= fLifterPosInUMToSltBtmMin(tylocalBuffer.In.diLifterCurrPosInUM , tylocalBuffer.In.diSltToSltInUM , tylocalBuffer.In.diLifterBtmPosInUM);

				IF tylocalBuffer.In.bNxtLoadSeq = TRUE THEN
					tylocalBuffer.Out.diNxtLoadSlt	:= fBffrNxtLoadSeqAny(tylocalBuffer.In.bAscending , tylocalBuffer.In.tylocalBuffer.Out.tyBuffer);
				ELSE
					tylocalBuffer.Out.diNxtLoadSlt	:= fBffrNxtLoadNearbyAny(tyLocalBuffer.Out.diCurrSlt , tylocalBuffer.In.tylocalBuffer.Out.tyBuffer);
				END_IF

				tylocalBuffer.Out.eStatus	:= Done;

			END_IF

		BufferActNxtLoadGd:
			IF tylocalBuffer.Out.eStatus = Idle OR tylocalBuffer.Out.eStatus = Busy THEN

				tyLocalBuffer.Out.diCurrSlt	:= fLifterPosInUMToSltBtmMin(tylocalBuffer.In.diLifterCurrPosInUM , tylocalBuffer.In.diSltToSltInUM , tylocalBuffer.In.diLifterBtmPosInUM);

				IF tylocalBuffer.In.bNxtLoadSeq = TRUE THEN
					tylocalBuffer.Out.diNxtLoadSlt	:= fBffrNxtLoadSeqGd(tylocalBuffer.In.bAscending , tylocalBuffer.In.tylocalBuffer.Out.tyBuffer);
				ELSE
					tylocalBuffer.Out.diNxtLoadSlt	:= fBffrNxtLoadNearbyGd(tyLocalBuffer.Out.diCurrSlt , tylocalBuffer.In.tylocalBuffer.Out.tyBuffer);
				END_IF

				tylocalBuffer.Out.eStatus	:= Done;

			END_IF

		BufferActNxtLoadBad:
			IF tylocalBuffer.Out.eStatus = Idle OR tylocalBuffer.Out.eStatus = Busy THEN

				tyLocalBuffer.Out.diCurrSlt	:= fLifterPosInUMToSltBtmMin(tylocalBuffer.In.diLifterCurrPosInUM , tylocalBuffer.In.diSltToSltInUM , tylocalBuffer.In.diLifterBtmPosInUM);

				IF tylocalBuffer.In.bNxtLoadSeq = TRUE THEN
					tylocalBuffer.Out.diNxtLoadSlt	:= fBffrNxtLoadSeqBad(tylocalBuffer.In.bAscending , tylocalBuffer.In.tylocalBuffer.Out.tyBuffer);
				ELSE
					tylocalBuffer.Out.diNxtLoadSlt	:= fBffrNxtLoadNearbyBad(tyLocalBuffer.Out.diCurrSlt , tylocalBuffer.In.tylocalBuffer.Out.tyBuffer);
				END_IF

				tylocalBuffer.Out.eStatus	:= Done;

			END_IF

		BufferActNxtUnload:
			IF tylocalBuffer.Out.eStatus = Idle OR tylocalBuffer.Out.eStatus = Busy THEN

				IF tylocalBuffer.In.bFIFO = TRUE THEN
					tylocalBuffer.Out.diNxtUnloadSlt	:= fBffrNxtUnloadFIFOAny(tylocalBuffer.In.tylocalBuffer.Out.tyBuffer , '');
				ELSE
					tylocalBuffer.Out.diNxtUnloadSlt	:= fBffrNxtUnloadLIFOAny(tylocalBuffer.In.tylocalBuffer.Out.tyBuffer , '');
				END_IF

				tylocalBuffer.Out.eStatus	:= Done;

			END_IF

		BufferActNxtUnloadGd:
			IF tylocalBuffer.Out.eStatus = Idle OR tylocalBuffer.Out.eStatus = Busy THEN

				IF tylocalBuffer.In.bFIFO = TRUE THEN
					tylocalBuffer.Out.diNxtUnloadSlt	:= fBffrNxtUnloadFIFOGd(tylocalBuffer.In.tylocalBuffer.Out.tyBuffer , '');
				ELSE
					tylocalBuffer.Out.diNxtUnloadSlt	:= fBffrNxtUnloadLIFOGd(tylocalBuffer.In.tylocalBuffer.Out.tyBuffer , '');
				END_IF

				tylocalBuffer.Out.eStatus	:= Done;

			END_IF

		BufferActNxtUnloadBad:
			IF tylocalBuffer.Out.eStatus = Idle OR tylocalBuffer.Out.eStatus = Busy THEN

				IF tylocalBuffer.In.bFIFO = TRUE THEN
					tylocalBuffer.Out.diNxtUnloadSlt	:= fBffrNxtUnloadFIFOBad(tylocalBuffer.In.tylocalBuffer.Out.tyBuffer , '');
				ELSE
					tylocalBuffer.Out.diNxtUnloadSlt	:= fBffrNxtUnloadLIFOBad(tylocalBuffer.In.tylocalBuffer.Out.tyBuffer , '');
				END_IF

				tylocalBuffer.Out.eStatus	:= Done;

			END_IF

		BufferActChkCoolTm:
			tyLocalBuffer.Out.diCurrSlt	:= fLifterPosInUMToSltBtmMin(tylocalBuffer.In.diLifterCurrPosInUM , tylocalBuffer.In.diSltToSltInUM , tylocalBuffer.In.diLifterBtmPosInUM);

			tylocalBuffer.Out.bCoolNotRdy	:= NOT fBffrChkCoolTmRdy(tyLocalBuffer.Out.diCurrSlt, tylocalBuffer.In.dtCurrDT, DINT_TO_TIME(tylocalBuffer.In.diCoolTm), tylocalBuffer.In.tylocalBuffer.Out.tyBuffer);

			tylocalBuffer.Out.eStatus	:= Done;

		BufferActChkCoolBrdAny:
			tylocalBuffer.Out.diCoolBrdAny	:= fBffrChkCoolBrdAny(tylocalBuffer.In.dtCurrDT, DINT_TO_TIME(tylocalBuffer.In.diCoolTm), tylocalBuffer.In.tylocalBuffer.Out.tyBuffer);

			tylocalBuffer.Out.eStatus	:= Done;

		BufferActChkCoolBrdGd:
			tylocalBuffer.Out.diCoolBrdGd		:= fBffrChkCoolBrdGd(tylocalBuffer.In.dtCurrDT, DINT_TO_TIME(tylocalBuffer.In.diCoolTm), tylocalBuffer.In.tylocalBuffer.Out.tyBuffer);

			tylocalBuffer.Out.eStatus	:= Done;

		BufferActChkCoolBrdBad:
			tylocalBuffer.Out.diCoolBrdBad	:= fBffrChkCoolBrdBad(tylocalBuffer.In.dtCurrDT, DINT_TO_TIME(tylocalBuffer.In.diCoolTm), tylocalBuffer.In.tylocalBuffer.Out.tyBuffer);

			tylocalBuffer.Out.eStatus	:= Done;

		BufferActRstBffr:
			IF tylocalBuffer.Out.eStatus = Idle OR tylocalBuffer.Out.eStatus = Busy THEN

				tyBffrParameter.diBffrTtlSlt	:= tylocalBuffer.In.diBffrTtlSlt;
				tyBffrParameter.diSltCap		:= tylocalBuffer.In.diSltCap;

				memset(ADR(tylocalBuffer.In.tylocalBuffer.Out.tyBuffer) , 0 , SIZEOF(tylocalBuffer.In.tylocalBuffer.Out.tyBuffer));
				fBffrStat(ADR(tylocalBuffer.In.tylocalBuffer.Out.tylocalBuffer.Out.tyBufferStat) , tylocalBuffer.In.tylocalBuffer.Out.tyBuffer);
				fDispBffrDescending(ADR(tylocalBuffer.In.tylocalBuffer.Out.tyDispBuffer) , tyBffrParameter , tylocalBuffer.In.tylocalBuffer.Out.tyBuffer , tylocalBuffer.In.dtCurrDT , DINT_TO_TIME(tylocalBuffer.In.diCoolTm) , 0 , 1 , 2);

				tylocalBuffer.Out.eStatus	:= Done;

			END_IF

		BufferActSetCoolFan:
			IF tylocalBuffer.Out.eStatus = Idle OR tylocalBuffer.Out.eStatus = Busy THEN

				tylocalBuffer.Out.bCoolFanCtrl	:= TRUE;
				tylocalBuffer.Out.eStatus			:= Done;

			END_IF

		BufferActRstCoolFan:
			IF tylocalBuffer.Out.eStatus = Idle OR tylocalBuffer.Out.eStatus = Busy THEN

				tylocalBuffer.Out.bCoolFanCtrl	:= FALSE;
				tylocalBuffer.Out.eStatus			:= Done;

			END_IF

		BufferActBGStartBffrSetFull:
			IF tylocalBuffer.Out.eStatus = Idle OR tylocalBuffer.Out.eStatus = Busy THEN

				bBffrSetFull	:= TRUE;
				bBffrSetMty		:= FALSE;
				tylocalBuffer.Out.eStatus			:= Done;

			END_IF

		BufferActBGStartBffrSetMty:
			IF tylocalBuffer.Out.eStatus = Idle OR tylocalBuffer.Out.eStatus = Busy THEN

				bBffrSetFull	:= FALSE;
				bBffrSetMty		:= TRUE;
				tylocalBuffer.Out.eStatus			:= Done;

			END_IF

		BufferActBGStopBffrSet:
			IF tylocalBuffer.Out.eStatus = Idle OR tylocalBuffer.Out.eStatus = Busy THEN

				bBffrSetFull	:= FALSE;
				bBffrSetMty		:= FALSE;
				tylocalBuffer.Out.eStatus			:= Done;

			END_IF

		BufferActBGStartUpdtSen:
			IF tylocalBuffer.Out.eStatus = Idle OR tylocalBuffer.Out.eStatus = Busy THEN

				bUpdateSensor	:= TRUE;
				tylocalBuffer.Out.eStatus			:= Done;

			END_IF

		BufferActBGStopUpdtSen:
			IF tylocalBuffer.Out.eStatus = Idle OR tylocalBuffer.Out.eStatus = Busy THEN

				bUpdateSensor	:= FALSE;
				tylocalBuffer.Out.eStatus			:= Done;

			END_IF

		BufferActBGStartUpdtDisplay:
			IF tylocalBuffer.Out.eStatus = Idle OR tylocalBuffer.Out.eStatus = Busy THEN

				bUpdtDisplay	:= TRUE;
				tylocalBuffer.Out.eStatus			:= Done;

			END_IF

		BufferActBGStopUpdtDisplay:
			IF tylocalBuffer.Out.eStatus = Idle OR tylocalBuffer.Out.eStatus = Busy THEN

				bUpdtDisplay	:= FALSE;
				tylocalBuffer.Out.eStatus			:= Done;

			END_IF

		BufferActBGStartCoolFan:
			IF tylocalBuffer.Out.eStatus = Idle OR tylocalBuffer.Out.eStatus = Busy THEN

				bCoolFanRun	:= TRUE;
				tylocalBuffer.Out.eStatus		:= Done;

			END_IF

		BufferActBGStopCoolFan:
			IF tylocalBuffer.Out.eStatus = Idle OR tylocalBuffer.Out.eStatus = Busy THEN

				bCoolFanRun	:= FALSE;
				tylocalBuffer.Out.eStatus		:= Done;

			END_IF

	END_CASE

END_ACTION
```

#### Act_Alarm.st - Do Not Change!!!
```iecst
(** 2019-03-25 **)
ACTION Act_Alarm:

	//Error
	IF EDGEPOS(eStatus = Error) THEN

		tyAlmData.sProgNm		:= p_sProgNm;
		tyAlmData.udiCode		:= udiStatus;
		tyAlmData.eSeverity		:= AlmSeverityError;
		tyAlmData.udiRunTime	:= tyAlmData.udiRunTime + 1;
		tyAlmData.bAlm			:= TRUE;
		tyAlmData.udiModuleNum  := udiModuleNum;
		g_sBufferProgNm		:= p_sProgNm;

		//Get Error Message
		IF tyAlmData.udiCode < 10000 OR tyAlmData.udiCode > 10099 THEN
			tyAlmData.sAlmMsg	:= 'Unknown';
			tyAlmData.sRcyMsg	:= 'Unknown';
		ELSE
			tyAlmData.sAlmMsg	:= a_tyAlmText[tyAlmData.udiCode].sAlmText;
			tyAlmData.sRcyMsg	:= a_tyAlmText[tyAlmData.udiCode].sRcyText;
		END_IF

		sStatTxt	:= tyAlmData.sAlmMsg;

	ELSIF bRstErr AND (tyAlmData.udiCode <> 0) THEN

		tyAlmData.udiCode	:= 0;
		tyAlmData.eSeverity	:= AlmSeverityNA;
		tyAlmData.sAlmMsg	:= '';
		tyAlmData.sRcyMsg	:= '';
		tyAlmData.bAlm			:= FALSE;
		sStatTxt	:= a_sStatText[eStat];

	END_IF

END_ACTION
```

#### Act_InputConfig.st - not listed in the package file held
```iecst
(** 2019-04-26 **)
ACTION Act_InputConfig:

	(* Always Change If Project Change *)

	//Pass Data To Link
	tylocalBuffer.In.bLinkPresentSen1 := g_tyDInput.bMagPresentSen2;
	tylocalBuffer.In.bLinkPresentSen2 := g_tyDInput.bMagConvEntSen2;
	tylocalBuffer.In.diLinkSltToSltDist ACCESS p_MagRcpCurrRcpSltToSlt;
	tylocalBuffer.In.bLinkMcParamProdSelTopToBtm ACCESS p_ProdRcpCurrRcp2TopToBtm;
	tylocalBuffer.In.bLinkOpsTravLifULExitBrd ACCESS p_OpsTravLifULExitBrd;

	//Pass Data To Internal Use
	tylocalBuffer.In.udiRstErr := g_tyRstErr.bReset;
	tylocalBuffer.In.sFileName := g_tyNtParamCurr.sBffr2FileNm;
	tylocalBuffer.In.bManual := g_tyUIOut.bManualMod;
	tylocalBuffer.In.dtCurrDT := g_tyTime.dtCurrDT;

	tylocalBuffer.In.diBffrTtlSlt ACCESS p_MagRcpCurrRcpTtlSlt;
	tylocalBuffer.In.diLifterBtmPosInUM ACCESS p_MagRcpCurrRcpMag2Slt1Pos;
	tylocalBuffer.In.diLifterCurrPosInUM := g_tyLifterBtm.diActualPos;
	tylocalBuffer.In.bGdBrdIn  := g_tyPshrConv.bGdBrd;
	tylocalBuffer.In.bNxtLoadSeq := g_tyNtParamCurr.bBffr2NxtLoadSeq;
	tylocalBuffer.In.sCurrRcpNm ACCESS p_ProdRcpCurrRcp2Nm;
	tylocalBuffer.In.sProgNm := g_tyNtParamCurr.sBffr2ProgNm;
	tylocalBuffer.In.bNtParamAutoRcpPrep := g_tyNtParamCurr.bAutoRcpPrep ;
	tylocalBuffer.In.bMcParamAutoRcpDis  := g_tyMcParamCurr.bAutoRcpDisable;

	//Siemens Req
	tylocalBuffer.In.bOpsMagConvULRlsMagAllw := g_tyOpsMagConvUL2.bRlsMagAllw;
	tylocalBuffer.In.eNtParamCustomerReq := g_tyNtParamCurr.eCustomerReq;
	tylocalBuffer.In.tyResponseFromMES :=  g_tyAGV.tyTagFromMesMagCov2;

	IF g_tyStartUp.bRun = TRUE THEN
		tylocalBuffer.In.eAct := g_tyStartUp.eBuffer2Act;
	ELSE
		IF tylocalBuffer.Out.eStatus = Idle THEN
			IF g_tyNtParamCurr.bProjLifterMagPlatform = FALSE THEN
				IF g_tyOpsMagConvUL2.eBufferAct <> BufferActIdle THEN
					tylocalBuffer.In.eAct := g_tyOpsMagConvUL2.eBufferAct;
				ELSIF g_tyUIOut.eBuffer2Act <> BufferActIdle THEN
					tylocalBuffer.In.eAct := g_tyUIOut.eBuffer2Act;
				ELSE
					tylocalBuffer.In.eAct := eAct;
				END_IF
			ELSE
				IF g_tyOpsLifMagULBufferAct2.eBufferAct <> BufferActIdle THEN
					tylocalBuffer.In.eAct := g_tyOpsLifMagULBufferAct2.eBufferAct;
				ELSE
					tylocalBuffer.In.eAct := g_tyUIOut.eBuffer2Act;
				END_IF
			END_IF
		END_IF
	END_IF

END_ACTION
```

#### Act_OutputConfig.st - not listed in the package file held
```iecst
(** 2019-06-07 **)
ACTION Act_OutputConfig:

	g_tyBuffer2 := tylocalBuffer.Out;

END_ACTION
```

### Program Logical/Buffer/Buffer3 (IEC, version 1.00.0) - 1.00.0 - NtBuffer v5.00.0 , NtFileIO v5.00.0

#### Init.st - Change By Project
```iecst
(** 2019-06-07 **)
PROGRAM _INIT

	(* Always Change If Project Change *)

	//Pass Address To Global Address For External Use
	//Action, State & Status
	p_Buffer3Stat		:= ADR(eStat);
	p_Buffer3Status		:= ADR(eStatus);
	p_Buffer3StatTxt	:= ADR(sStatTxt);

	//Alarm
	p_Buffer3AlmData	:= ADR(tyAlmData);

	//Output
	p_Buffer3NxtLoadSlt				:= ADR(diNxtLoadSlt);
	p_Buffer3NxtUnloadSlt			:= ADR(diNxtUnloadSlt);
	p_Buffer3CoolBrdAny				:= ADR(diCoolBrdAny);
	p_Buffer3CoolBrdGd				:= ADR(diCoolBrdGd);
	p_Buffer3CoolBrdBad				:= ADR(diCoolBrdBad);
	p_Buffer3CoolNotRdy				:= ADR(bCoolNotRdy);
	p_Buffer3Bffr					:= ADR(tyBuffer);
	p_Buffer3DispBffr				:= ADR(tyDispBuffer);
	p_Buffer3BffrStat				:= ADR(tyBufferStat);
	p_Buffer3BrdUnloadStat			:= ADR(tyBoardUnloadStat);
	p_Buffer3FileNotFound			:= ADR(bFileNotFound);
	p_Buffer3CoolFanCtrl			:= ADR(bCoolFanCtrl);
	p_Buffer3MagPresent				:= ADR(bMagPresent);
	p_Buffer3MagPresentTm			:= ADR(dtMagPresentTm);
	p_Buffer3NewProduct				:= ADR(bNewProduct);
	p_Buffer3LastProductUnload		:= ADR(bLastProductUnload);
	p_Buffer3LastProductLeftInBffr	:= ADR(bLastProductLeftInBffr);
	p_Buffer3ParamDiff				:= ADR(bParamDiff);
	p_Buffer3MagRemoved				:= ADR(bMagRemoved);
	p_Buffer3FIFOOld				:= ADR(bFIFOOld);

	//Svy Hermes
	p_Buffer3SlotNo					:= ADR(diCurrSlt);
	(* Always Change If Project Change *)

END_PROGRAM
```

#### Act_InitGlobal.st - Change By Project
```iecst
(** 2019-04-26 **)
ACTION Act_InitGlobal:

	(* Always Change If Project Change *)

	//Pass Data To Link
	p_bLinkStartupRun ACCESS p_StartupRun;
	p_bLinkNtParamProjMagConvPrep ACCESS p_NtParamProjMag3ConvPrep;
//	p_eLinkOpsMagULBufferAct ACCESS p_OpsMagUL3BufferAct;
	p_eLinkOpsMagConvULBufferAct ACCESS p_OpsMagConvUL3BufferAct;
	p_eLinkUIBufferAct ACCESS p_UIBuffer3Act;
	p_bLinkProjLifterMagPlatform ACCESS p_NtParamProjLifterMagPlatform;
	p_eLinkOpsLifMagULBufferAct ACCESS p_OpsLifMagULBufferAct3;

	p_diLinkSltToSltDist ACCESS p_MagRcpCurrRcpSltToSlt;
	p_bLinkMcParamProdSelTopToBtm ACCESS p_ProdRcpCurrRcp2TopToBtm;
	p_bLinkPresentSen1 ACCESS p_DIMagPresentSen3;
	p_bLinkPresentSen2 ACCESS p_DIMagConvEntSen3;
	p_bLinkOpsTravLifULExitBrd ACCESS p_OpsTravLifULExitBrd;

	//Pass Data To Internal Use
	p_udiRstErr ACCESS p_RstErrReset;
	p_sFileName ACCESS p_NtParamBffr3FileNm;
	p_bManual ACCESS p_UIMnlMod;
	p_dtCurrDT ACCESS p_TimeCurrDT;

	p_diBffrTtlSlt ACCESS p_MagRcpCurrRcpTtlSlt;
	p_diLifterBtmPosInUM ACCESS p_MagRcpCurrRcpMag3Slt1Pos;
	p_diLifterCurrPosInUM ACCESS p_LifterBtmActualPos;
	p_bGdBrdIn ACCESS p_PshrConvGdBrd;
	p_bNxtLoadSeq ACCESS p_NtParamBffr3NxtLoadSeq;
//	p_bMagPresentSensor ACCESS p_DIMagPresentSen3;
	p_sCurrRcpNm ACCESS p_ProdRcpCurrRcp2Nm;
	p_sProgNm ACCESS p_NtParamBffr3ProgNm;
	p_bNtSettingsLoadDone ACCESS p_StartupNtSettingsLoadDone;
	p_bNtParamAutoRcpPrep ACCESS p_NtParamAutoRcpPrep ;
	p_bMcParamAutoRcpDis  ACCESS p_McParamAutoRcpDisable;

	//Siemens Req
	p_bOpsMagConvULRlsMagAllw ACCESS p_OpsMagConvUL3RlsMagAllw;
	p_eNtParamCustomerReq ACCESS p_NtParamCustomerReq;
	p_tyResponseFromMES ACCESS p_TagFromMesMagConv3; //Siemens Req

	p_bNtParamAutoRcpF1ArbitraryType ACCESS p_NtParamAutoRcpF1ArbitraryType;
	(* Always Change If Project Change *)

END_ACTION
```

#### InputRef_Link.var - Change By Project
```iecst
(*2019-04-09*)
(**)
(*External*)
VAR
	p_bLinkStartupRun : REFERENCE TO BOOL;
	p_bLinkNtParamProjMagConvPrep : REFERENCE TO BOOL;
	p_eLinkOpsMagULBufferAct : REFERENCE TO eBufferAction;
	p_eLinkOpsMagConvULBufferAct : REFERENCE TO eBufferAction;
	p_eLinkUIBufferAct : REFERENCE TO eBufferAction;
END_VAR
(**)
VAR
	p_diLinkSltToSltDist : REFERENCE TO DINT;
	p_bLinkMcParamProdSelTopToBtm : REFERENCE TO BOOL;
	p_bLinkPresentSen1 : REFERENCE TO BOOL;
	p_bLinkPresentSen2 : REFERENCE TO BOOL;
	p_bLinkProjLifterMagPlatform : REFERENCE TO BOOL;
	p_eLinkOpsLifMagULBufferAct : REFERENCE TO eBufferAction;
	p_bLinkOpsTravLifULExitBrd : REFERENCE TO BOOL;
END_VAR
```

#### Act_LinkAction.st - Change By Project
```iecst
(** 2019-05-10 **)
ACTION Act_LinkAction:

	IF p_bLinkStartupRun = TRUE THEN
		p_eAct ACCESS p_StartupBuffer3Act;
	ELSE
		IF eStatus = Idle THEN
			IF p_bLinkProjLifterMagPlatform = FALSE THEN
				IF p_eLinkOpsMagConvULBufferAct <> BufferActIdle THEN
					p_eAct ACCESS p_OpsMagConvUL3BufferAct;
				ELSIF p_eLinkUIBufferAct <> BufferActIdle THEN
					p_eAct ACCESS p_UIBuffer3Act;
				ELSE
					p_eAct ACCESS ADR(eAct);
				END_IF
			ELSE
				IF p_eLinkOpsLifMagULBufferAct <> BufferActIdle THEN
					p_eAct ACCESS p_OpsLifMagULBufferAct3;
				ELSE
					p_eAct ACCESS p_UIBuffer3Act;
				END_IF
			END_IF
		END_IF
	END_IF

END_ACTION
```

#### Act_Link.st - Change By Project
```iecst
(** 2019-03-29 **)
ACTION Act_Link:
	IF g_tyNtParamCurr.bAutoRcpPrep AND NOT(g_tyMcParamCurr.bAutoRcpDisable) THEN
		tylocalBuffer.In.diMinSlt ACCESS g_tyAutoRcpMag3.diMinSlt;
		tylocalBuffer.In.diMaxSlt ACCESS g_tyAutoRcpMag3.diMaxSlt;
		tylocalBuffer.In.diPitch ACCESS g_tyAutoRcpMag3.diPitch;
	ELSE
		tylocalBuffer.In.diMinSlt ACCESS p_ProdRcpCurrRcp2MinSltValue;
		tylocalBuffer.In.diMaxSlt ACCESS p_ProdRcpCurrRcp2MaxSltValue;
		tylocalBuffer.In.diPitch ACCESS p_ProdRcpCurrRcp2Pitch;
	END_IF
	IF g_tyNtParamCurr.bProjLifterMagPlatform THEN
		tylocalBuffer.In.diSltToSltInUM ACCESS p_MagRcpCurrRcpSltToSlt;
	ELSE
		tylocalBuffer.In.diSltToSltInUM	:= tylocalBuffer.In.diLinkSltToSltDist * -1;
	END_IF

	tylocalBuffer.In.bAscending	:= NOT tylocalBuffer.In.bLinkMcParamProdSelTopToBtm;

	IF tylocalBuffer.In.bLinkOpsTravLifULExitBrd THEN
		tylocalBuffer.In.bMagPresentSensor := tylocalBuffer.In.bLinkPresentSen1; //present sensor only
	ELSE
		tylocalBuffer.In.bMagPresentSensor := tylocalBuffer.In.bLinkPresentSen1 OR tylocalBuffer.In.bLinkPresentSen2;
	END_IF

	//For MES Call Full
	IF tylocalBuffer.In.tyResponseFromMES.bTrigMagFull AND tylocalBuffer.In.bOpsMagConvULRlsMagAllw
		AND NOT(tylocalBuffer.Out.tyBufferStat.bBffrFull)  AND tylocalBuffer.In.eNtParamCustomerReq = Siemens THEN
		bMESTrigSetFull	:= TRUE;
	END_IF
	IF bMESTrigSetFull THEN
		tylocalBuffer.In.eAct	:= BufferActSetFull;
		IF tylocalBuffer.Out.eStat = BufferActSetFull AND tylocalBuffer.Out.eStatus = Done THEN
			tylocalBuffer.In.eAct	:= BufferActIdle;
			bMESTrigSetFull := FALSE;
		END_IF
	END_IF
END_ACTION
```

#### Cyclic.st - Do Not Change!!!
```iecst
(** 2019-03-29 **)
PROGRAM _CYCLIC

	IF bInitialDone = FALSE THEN
		IF g_tyStartUp.bNtSettingsLoadDone = TRUE THEN
			bInitialDone	:= TRUE;
			Act_Initial;
		END_IF

	ELSE
		Act_InputConfig
		Act_Link;
		Act_Main;
		Act_OutputConfig;
		Act_Alarm;
	END_IF

END_PROGRAM
```

#### Act_Initial.st - Do Not Change!!!
```iecst
(** 2019-04-26 **)
ACTION Act_Initial:

	//Initial
	tylocalBuffer.Out.sStatTxt	:= a_sStatText[eStat];

	fbDirCreate1.sDevice	:= 'F';
	fbDirCreate1.sDirName	:= 'User';
	fbDirCreate1(bEn := FALSE);

	fbDirCreate2.sDevice	:= 'User';
	fbDirCreate2.sDirName	:= 'Retain';
	fbDirCreate2(bEn := FALSE);

	fbFileRead1.sDevice			:= 'Retain';
	fbFileRead1.sFile			:= tylocalBuffer.In.sFileName;
	fbFileRead1.udiOffset		:= 0;
	fbFileRead1.p_Dest			:= ADR(tylocalBuffer.In.tyBuffer);
	fbFileRead1.udiLen			:= SIZEOF(tylocalBuffer.In.tyBuffer);
	fbFileRead1(bEn := FALSE);

	fbFileWrite1.sDevice		:= 'Retain';
	fbFileWrite1.sFile			:= tylocalBuffer.In.sFileName;
	fbFileWrite1.udiOffset		:= 0;
	fbFileWrite1.p_Src			:= ADR(tylocalBuffer.In.tyBuffer);
	fbFileWrite1.udiLen			:= SIZEOF(tylocalBuffer.In.tyBuffer);
	fbFileWrite1.udiOption		:= 0;
	fbFileWrite1(bEn := FALSE);

	fbCoolFanOffDlyTm.PT	:= DINT_TO_TIME(tylocalBuffer.In.diCoolFanOffDlyTm);
	fbCoolFanOffDlyTm(IN := FALSE);

	fbCoolFanOffChkTm(IN := FALSE);
	fbMagAbsentTm(IN := FALSE);
	fbMagPresentTm(IN := FALSE);

END_ACTION
```

#### Act_Alarm.st - Do Not Change!!!
```iecst
(** 2019-03-25 **)
ACTION Act_Alarm:
	IF tylocalBuffer.In.udiRstErr <> udiRstErrOld THEN
		bRstErr			:= TRUE;
		udiRstErrOld	:= tylocalBuffer.In.udiRstErr;
	ELSE
		bRstErr			:= FALSE;
	END_IF
	//Reset Error
	IF (tylocalBuffer.Out.eStatus = Error) AND bRstErr THEN
		tylocalBuffer.In.eAct	:= BufferActIdle;
		tylocalBuffer.Out.eStat	:= BufferActIdle;
	END_IF
	//Error
	IF EDGEPOS(tylocalBuffer.Out.eStatus = Error) THEN

		tylocalBuffer.Out.tyAlmData.sProgNm		:= tylocalBuffer.In.sProgNm;
		tylocalBuffer.Out.tyAlmData.udiCode		:= udiStatus;
		tylocalBuffer.Out.tyAlmData.eSeverity		:= AlmSeverityError;
		tylocalBuffer.Out.tyAlmData.udiRunTime	:= tylocalBuffer.Out.tyAlmData.udiRunTime + 1;
		tylocalBuffer.Out.tyAlmData.bAlm			:= TRUE;
		tylocalBuffer.Out.tyAlmData.udiModuleNum  := udiModuleNum;
		g_sBufferProgNm			:= tylocalBuffer.In.sProgNm;

		tylocalBuffer.Out.sStatTxt	:= tylocalBuffer.Out.tyAlmData.sAlmMsg;

	ELSIF bRstErr AND (tylocalBuffer.Out.tyAlmData.udiCode <> 0) THEN

		tylocalBuffer.Out.tyAlmData.udiCode	:= 0;
		tylocalBuffer.Out.tyAlmData.eSeverity	:= AlmSeverityNA;

		tylocalBuffer.Out.tyAlmData.bAlm			:= FALSE;
		tylocalBuffer.Out.sStatTxt	:= a_sStatText[tylocalBuffer.Out.eStat];

	END_IF

END_ACTION
```

#### InputRef.var - Do Not Change!!!
```iecst
(*2019-07-03*)
(**)
(*General*)
VAR
	p_eAct : REFERENCE TO eBufferAction;
	p_udiRstErr : REFERENCE TO UDINT;
END_VAR
(**)
(*Configuration*)
VAR
	p_sFileName : REFERENCE TO STRING[80];
	p_bManual : REFERENCE TO BOOL;
	p_dtCurrDT : REFERENCE TO DATE_AND_TIME;
	p_diMinSlt : REFERENCE TO DINT;
	p_diMaxSlt : REFERENCE TO DINT;
	p_diPitch : REFERENCE TO DINT;
	p_diSltCap : REFERENCE TO DINT;
	p_diBffrTtlSlt : REFERENCE TO DINT;
	p_diCoolTm : REFERENCE TO DINT;
	p_diSltToSltInUM : REFERENCE TO DINT;
	p_diLifterBtmPosInUM : REFERENCE TO DINT;
	p_diLifterCurrPosInUM : REFERENCE TO DINT;
	p_bAscending : REFERENCE TO BOOL;
	p_bFIFO : REFERENCE TO BOOL;
	p_bGdBrdIn : REFERENCE TO BOOL;
	p_bGdBrdReq : REFERENCE TO BOOL;
	p_bNxtLoadSeq : REFERENCE TO BOOL;
	pa_bSkip : REFERENCE TO ARRAY[1..c_diBffrSize] OF BOOL;
	p_diCoolFanOffDlyTm : REFERENCE TO DINT;
	p_bMagPresentSensor : REFERENCE TO BOOL;
	p_bPrepCoolFan : REFERENCE TO BOOL;
	p_bCoolFanTm : REFERENCE TO BOOL;
	p_tyBuffer : REFERENCE TO tyBffr;
	p_tyDispBuffer : REFERENCE TO tyDispBffr;
	p_tyBufferStat : REFERENCE TO tyBffrStat;
	p_sBffrNm : REFERENCE TO STRING[15];
	p_sProdNm : REFERENCE TO STRING[15];
	p_sBarcode1 : REFERENCE TO STRING[80];
	p_sBarcode2 : REFERENCE TO STRING[80];
	p_sCurrRcpNm : REFERENCE TO STRING[15];
	p_sProgNm : REFERENCE TO STRING[15];
	p_bNtSettingsLoadDone : REFERENCE TO BOOL;
	p_bNtParamAutoRcpPrep : REFERENCE TO BOOL;
	p_bMcParamAutoRcpDis : REFERENCE TO BOOL;
	p_bOpsMagConvULRlsMagAllw : REFERENCE TO BOOL;
	p_eNtParamCustomerReq : REFERENCE TO eCustomer;
	p_tyResponseFromMES1 : REFERENCE TO tyStatPlatformFromMES;
	p_bNtParamAutoRcpF1ArbitraryType : REFERENCE TO BOOL;
	p_tyResponseFromMES : REFERENCE TO tyStatPlatformFromMES;
END_VAR
```

#### Local.var - Do Not Change!!!
```iecst
(*2019-06-07*)
(**)
(*Local Action, State & Status*)
VAR
	tylocalBuffer : tyBuffer1;
	eAct : eBufferAction := BufferActIdle;
	udiStatus : UDINT := 0;
	a_sStatText : ARRAY[0..50] OF STRING[200] := ['Idling','Creating Directory','Getting Retained Buffer Data','Setting Buffer Full','Setting Buffer Empty','Loading Board','Loading Board With Slot Check','Unloading Board','Unloading Board With Slot Check','Unloading Board With Cooling Time Check','Unloading Board With Slot Check And Cooling Time Check','Getting Next Load Board Slot Number','Getting Next Load Good Board Slot Number','Getting Next Load Bad Board Slot Number','Getting Next Unload Board Slot Number','Getting Next Unload Good Board Slot Number','Getting Next Unload Bad Board Slot Number','Checking Cooling Time','Checking Cooling Board','Checking Cooling Good Board','Checking Cooling Bad Board','Resetting Buffer','Turning On Cooling Fan','Turning Off Cooling Fan','Background Starting Buffer Set Full','Background Starting Buffer Set Empty','Background Stopping Buffer Set','Background Starting Update Sensor','Background Stopping Update Sensor','Background Starting Update Display','Background Stopping Update Display','Background Starting Cooling Fan','Background Stopping Cooling Fan',18('')];
END_VAR
(**)
(*Local Alarm*)
VAR
	tyAlmData : tyAlmDat;
	a_tyAlmText : ARRAY[10000..10099] OF tyAlmTxt := [(sAlmText:='Create User Directory Error',sRcyText:='An Error Occurred While Attempting To Create User Directory. Please Contact Nutek For A Possible Solution'),(sAlmText:='Create Retain Directory Error',sRcyText:='An Error Occurred While Attempting To Create Retain Directory. Please Contact Nutek For A Possible Solution'),(sAlmText:='File Open Error While Reading Retain File',sRcyText:='An Error Was Encountered While Trying To Open File. Please Contact Nutek For A Possible Solution.'),(sAlmText:='File Read Error While Reading Retain File',sRcyText:='An Error Was Encountered While Trying To Read File. Please Contact Nutek For A Possible Solution.'),(sAlmText:='File Close Error While Reading Retain File',sRcyText:='An Error Was Encountered While Trying To Close File. Please Contact Nutek For A Possible Solution.'),(sAlmText:='File Open Error While Setting Full Buffer',sRcyText:='An Error Was Encountered While Trying To Open File. Please Contact Nutek For A Possible Solution.'),(sAlmText:='File Create Error While Setting Full Buffer',sRcyText:='An Error Was Encountered While Trying To Create File. Please Contact Nutek For A Possible Solution.'),(sAlmText:='File Write Error While Setting Full Buffer',sRcyText:='An Error Was Encountered While Trying To Write File. Please Contact Nutek For A Possible Solution.'),(sAlmText:='File Close Error While Setting Full Buffer',sRcyText:='An Error Was Encountered While Trying To Close File. Please Contact Nutek For A Possible Solution.'),(sAlmText:='File Open Error While Setting Empty Buffer',sRcyText:='An Error Was Encountered While Trying To Open File. Please Contact Nutek For A Possible Solution.'),(sAlmText:='File Create Error While Setting Empty Buffer',sRcyText:='An Error Was Encountered While Trying To Create File. Please Contact Nutek For A Possible Solution.'),(sAlmText:='File Write Error While Setting Empty Buffer',sRcyText:='An Error Was Encountered While Trying To Write File. Please Contact Nutek For A Possible Solution.'),(sAlmText:='File Close Error While Setting Empty Buffer',sRcyText:='An Error Was Encountered While Trying To Close File. Please Contact Nutek For A Possible Solution.'),(sAlmText:='File Open Error While Loading Info To Buffer',sRcyText:='An Error Was Encountered While Trying To Open File. Please Contact Nutek For A Possible Solution.'),(sAlmText:='File Create Error While Loading Info To Buffer',sRcyText:='An Error Was Encountered While Trying To Create File. Please Contact Nutek For A Possible Solution.'),(sAlmText:='File Write Error While Loading Info To Buffer',sRcyText:='An Error Was Encountered While Trying To Write File. Please Contact Nutek For A Possible Solution.'),(sAlmText:='File Close Error While Loading Info To Buffer',sRcyText:='An Error Was Encountered While Trying To Close File. Please Contact Nutek For A Possible Solution.'),(sAlmText:='Wrong Slot Number To Load',sRcyText:='Invalid Slot to Load The Board.'),(sAlmText:='File Open Error While Loading Info To Buffer With Slot Check',sRcyText:='An Error Was Encountered While Trying To Open File. Please Contact Nutek For A Possible Solution.'),(sAlmText:='File Create Error While Loading Info To Buffer With Slot Check',sRcyText:='An Error Was Encountered While Trying To Create File. Please Contact Nutek For A Possible Solution.'),(sAlmText:='File Write Error While Loading Info To Buffer With Slot Check',sRcyText:='An Error Was Encountered While Trying To Write File. Please Contact Nutek For A Possible Solution.'),(sAlmText:='File Close Error While Loading Info To Buffer With Slot Check',sRcyText:='An Error Was Encountered While Trying To Close File. Please Contact Nutek For A Possible Solution.'),(sAlmText:='File Open Error While Unloading Info From Buffer',sRcyText:='An Error Was Encountered While Trying To Open File. Please Contact Nutek For A Possible Solution.'),(sAlmText:='File Create Error While Unloading Info From Buffer',sRcyText:='An Error Was Encountered While Trying To Create File. Please Contact Nutek For A Possible Solution.'),(sAlmText:='File Write Error While Unloading Info From Buffer',sRcyText:='An Error Was Encountered While Trying To Write File. Please Contact Nutek For A Possible Solution.'),(sAlmText:='File Close Error While Unloading Info From Buffer',sRcyText:='An Error Was Encountered While Trying To Close File. Please Contact Nutek For A Possible Solution.'),(sAlmText:='Wrong Slot Number To Unload',sRcyText:='Invalid Slot to Unload The Board.'),(sAlmText:='File Open Error While Unloading Info From Buffer With Slot Check',sRcyText:='An Error Was Encountered While Trying To Open File. Please Contact Nutek For A Possible Solution.'),(sAlmText:='File Create Error While Unloading Info From Buffer With Slot Check',sRcyText:='An Error Was Encountered While Trying To Create File. Please Contact Nutek For A Possible Solution.'),(sAlmText:='File Write Error While Unloading Info From Buffer With Slot Check',sRcyText:='An Error Was Encountered While Trying To Write File. Please Contact Nutek For A Possible Solution.'),(sAlmText:='File Close Error While Unloading Info From Buffer With Slot Check',sRcyText:='An Error Was Encountered While Trying To Close File. Please Contact Nutek For A Possible Solution.'),(sAlmText:='File Open Error While Unloading Info From Buffer With Cooling Time Check',sRcyText:='An Error Was Encountered While Trying To Open File. Please Contact Nutek For A Possible Solution.'),(sAlmText:='File Create Error While Unloading Info From Buffer With Cooling Time Check',sRcyText:='An Error Was Encountered While Trying To Create File. Please Contact Nutek For A Possible Solution.'),(sAlmText:='File Write Error While Unloading Info From Buffer With Cooling Time Check',sRcyText:='An Error Was Encountered While Trying To Write File. Please Contact Nutek For A Possible Solution.'),(sAlmText:='File Close Error While Unloading Info From Buffer With Cooling Time Check',sRcyText:='An Error Was Encountered While Trying To Close File. Please Contact Nutek For A Possible Solution.'),(sAlmText:='Wrong Slot Number To Unload With Cooling Time Check',sRcyText:='Invalid Slot to Unload The Board with Cooling Time Check.'),(sAlmText:='File Open Error While Unloading Info From Buffer With Slot Check And Cooling Time Check',sRcyText:='An Error Was Encountered While Trying To Open File. Please Contact Nutek For A Possible Solution.'),(sAlmText:='File Create Error While Unloading Info From Buffer With Slot Check And Cooling Time Check',sRcyText:='An Error Was Encountered While Trying To Create File. Please Contact Nutek For A Possible Solution.'),(sAlmText:='File Write Error While Unloading Info From Buffer With Slot Check And Cooling Time Check',sRcyText:='An Error Was Encountered While Trying To Write File. Please Contact Nutek For A Possible Solution.'),(sAlmText:='File Close Error While Unloading Info From Buffer With Slot Check And Cooling Time Check',sRcyText:='An Error Was Encountered While Trying To Close File. Please Contact Nutek For A Possible Solution.'),(sAlmText:='Directory Does Not Exist While Setting Full Buffer',sRcyText:='The Directory Does Not Exist. Please Contact Nutek For A Possible Solution.'),(sAlmText:='Directory Does Not Exist While Setting Empty Buffer',sRcyText:='The Directory Does Not Exist. Please Contact Nutek For A Possible Solution.'),(sAlmText:='Directory Does Not Exist While Loading Info To Buffer',sRcyText:='The Directory Does Not Exist. Please Contact Nutek For A Possible Solution.'),(sAlmText:='Directory Does Not Exist While Loading Info To Buffer With Slot Check',sRcyText:='The Directory Does Not Exist. Please Contact Nutek For A Possible Solution.'),(sAlmText:='Directory Does Not Exist While Unloading Info From Buffer',sRcyText:='The Directory Does Not Exist. Please Contact Nutek For A Possible Solution.'),(sAlmText:='Directory Does Not Exist While Unloading Info From Buffer With Slot Check',sRcyText:='The Directory Does Not Exist. Please Contact Nutek For A Possible Solution.'),(sAlmText:='Directory Does Not Exist While Unloading Info From Buffer With Cooling Time Check',sRcyText:='The Directory Does Not Exist. Please Contact Nutek For A Possible Solution.'),(sAlmText:='Directory Does Not Exist While Unloading Info From Buffer With Slot Check And Cooling Time Check',sRcyText:='The Directory Does Not Exist. Please Contact Nutek For A Possible Solution.'),(sAlmText:='Unloading Slot Is Skipped While Unloading Buffer',sRcyText:='Unload From Wrong Slot (Skip Slot).'),(sAlmText:='Unloading Slot Is Not For Board While Unloading Buffer',sRcyText:='Unload From Wrong Slot (Not For Board).'),(sAlmText:='Unloading Slot Board Is Not Available While Unloading Buffer',sRcyText:='Unload From Wrong Slot (Board Is Not Available).'),(sAlmText:='Unloading Last Sub Slot Is Not For Board While Unloading Buffer',sRcyText:='Unload From Wrong Slot (Last Sub Slot Is Not For Board).'),(sAlmText:='Unloading Last Sub Slot Has No Board While Unloading Buffer',sRcyText:='Unload From Wrong Slot (Last Sub Slot Has No Board).'),(sAlmText:='Board Quantity In Slot Is 0 While Unloading Buffer',sRcyText:='Unload From Wrong Slot (Board Quantity In Slot = 0).'),(sAlmText:='Board Capacity In Slot Is 0 While Unloading Buffer',sRcyText:='Unload From Wrong Slot (Board Capacity In Slot = 0).'),(sAlmText:='Unloading Slot Is Skipped While Unloading Buffer With Slot Check',sRcyText:='Unload From Wrong Slot (Skip Slot).'),(sAlmText:='Unloading Slot Is Not For Board While Unloading Buffer With Slot Check',sRcyText:='Unload From Wrong Slot (Not For Board).'),(sAlmText:='Unloading Slot Board Is Not available While Unloading Buffer With Slot Check',sRcyText:='Unload From Wrong Slot (Board Is Not Available).'),(sAlmText:='Unloading Last Sub Slot Is Not For Board While Unloading Buffer With Slot Check',sRcyText:='Unload From Wrong Slot (Last Sub Slot Is Not For Board).'),(sAlmText:='Unloading Last Sub Slot Has No Board While Unloading Buffer With Slot Check',sRcyText:='Unload From Wrong Slot (Last Sub Slot Has No Board).'),(sAlmText:='Board Quantity In Slot Is 0 While Unloading Buffer With Slot Check',sRcyText:='Unload From Wrong Slot (Board Quantity In Slot = 0).'),(sAlmText:='Board Capacity In Slot Is 0 While Unloading Buffer With Slot Check',sRcyText:='Unload From Wrong Slot (Board Capacity In Slot = 0).'),(sAlmText:='Unloading Slot Is Skipped While Unloading Buffer With Cool Check',sRcyText:='Unload From Wrong Slot (Skip Slot).'),(sAlmText:='Unloading Slot Is Not For Board While Unloading Buffer With Cool Check',sRcyText:='Unload From Wrong Slot (Not For Board).'),(sAlmText:='Unloading Slot Board Is Not available While Unloading Buffer With Cool Check',sRcyText:='Unload From Wrong Slot (Board Is Not Available).'),(sAlmText:='Unloading Last Sub Slot Is Not For Board While Unloading Buffer With Cool Check',sRcyText:='Unload From Wrong Slot (Last Sub Slot Is Not For Board).'),(sAlmText:='Unloading Last Sub Slot Has No Board While Unloading Buffer With Cool Check',sRcyText:='Unload From Wrong Slot (Last Sub Slot Has No Board).'),(sAlmText:='Board Quantity In Slot Is 0 While Unloading Buffer With Cool Check',sRcyText:='Unload From Wrong Slot (Board Quantity In Slot = 0).'),(sAlmText:='Board Capacity In Slot Is 0 While Unloading Buffer With Cool Check',sRcyText:='Unload From Wrong Slot (Board Capacity In Slot = 0).'),(sAlmText:='Unloading Slot Is Skipped While Unloading Buffer With Cool & Slot Check',sRcyText:='Unload From Wrong Slot (Skip Slot).'),(sAlmText:='Unloading Slot Is Not For Board While Unloading Buffer With Cool & Slot Check',sRcyText:='Unload From Wrong Slot (Not For Board).'),(sAlmText:='Unloading Slot Board Is Not available While Unloading Buffer With Cool & Slot Check',sRcyText:='Unload From Wrong Slot (Board Is Not Available).'),(sAlmText:='Unloading Last Sub Slot Is Not For Board While Unloading Buffer With Cool & Slot Check',sRcyText:='Unload From Wrong Slot (Last Sub Slot Is Not For Board).'),(sAlmText:='Unloading Last Sub Slot Has No Board While Unloading Buffer With Cool & Slot Check',sRcyText:='Unload From Wrong Slot (Last Sub Slot Has No Board).'),(sAlmText:='Board Quantity In Slot Is 0 While Unloading Buffer With Cool & Slot Check',sRcyText:='Unload From Wrong Slot (Board Quantity In Slot = 0).'),(sAlmText:='Board Capacity In Slot Is 0 While Unloading Buffer With Cool & Slot Check',sRcyText:='Unload From Wrong Slot (Board Capacity In Slot = 0).'),(sAlmText:='Loading Slot Is Not For Board',sRcyText:='Load To Wrong Slot (Not For Board).'),(sAlmText:='Loading Slot Is Full Of Board',sRcyText:='Load To Wrong Slot (Full With Board).'),(sAlmText:='Loading First Sub-Slot Is Not For Board',sRcyText:='Load To Wrong Slot (First Sub Slot Not For Board).'),(sAlmText:='Loading Last Sub-Slot Have Board, Which Mean Slot Is Full Of Board',sRcyText:='Load To Wrong Slot (Full With Board(Last Sub Slot Have Board)).'),(sAlmText:='Loading Last Sub-Slot Is Not For Board',sRcyText:='Load To Wrong Slot (Last Sub Slot Not For Board).'),(sAlmText:='Loading Slot Is Full Of Board',sRcyText:='Load To Wrong Slot (Full With Board).'),(sAlmText:='Loading Slot Is Skipped',sRcyText:='Load To Wrong Slot (Skip Slot).'),(sAlmText:='Existing Board Status Is Different With Loading Board Status',sRcyText:='Existing Board Status Is Different With Loading Buffer Status.'),(sAlmText:='Loading Slot Is Not For Board',sRcyText:='Load To Wrong Slot (Not For Board).'),(sAlmText:='Loading Slot Is Full Of Board',sRcyText:='Load To Wrong Slot (Full With Board).'),(sAlmText:='Loading First Sub-Slot Is Not For Board',sRcyText:='Load To Wrong Slot (First Sub Slot Not For Board).'),(sAlmText:='Loading Last Sub-Slot Have Board, Which Mean Slot Is Full Of Board',sRcyText:='Load To Wrong Slot (Full With Board(Last Sub Slot Have Board)).'),(sAlmText:='Loading Last Sub-Slot Is Not For Board',sRcyText:='Load To Wrong Slot (Last Sub Slot Not For Board).'),(sAlmText:='Loading Slot Is Full Of Board',sRcyText:='Load To Wrong Slot (Full With Board).'),(sAlmText:='Loading Slot Is Skipped',sRcyText:='Load To Wrong Slot (Skip Slot).'),(sAlmText:='Existing Board Status Is Different With Loading Board Status',sRcyText:='Existing Board Status Is Different With Loading Buffer Status.'),8((0))];
END_VAR
(**)
(**)
(*Local Input*)
VAR
	udiRstErr : UDINT := 0;
	sFileName : STRING[80] := 'Buffer.dat';
	bManual : BOOL := FALSE;
	dtCurrDT : DATE_AND_TIME;
	diMinSlt : DINT;
	diMaxSlt : DINT;
	diPitch : DINT;
	diSltCap : DINT := 1;
	diBffrTtlSlt : DINT;
	diCoolTm : DINT;
	diSltToSltInUM : DINT;
	diLifterBtmPosInUM : DINT;
	diLifterCurrPosInUM : DINT;
	bAscending : BOOL;
	bFIFO : BOOL;
	bGdBrdIn : BOOL;
	bGdBrdReq : BOOL;
	bNxtLoadSeq : BOOL;
	a_bSkip : ARRAY[1..c_diBffrSize] OF BOOL;
	diCoolFanOffDlyTm : DINT := 30000;
	bMagPresentSensor : BOOL;
	bPrepCoolFan : BOOL := TRUE;
	bCoolFanTm : BOOL := TRUE;
	sBffrNm : STRING[15];
	sProdNm : STRING[15];
	sBarcode1 : STRING[80];
	sBarcode2 : STRING[80];
	sCurrRcpNm : {REDUND_UNREPLICABLE} STRING[15];
	sProgNm : STRING[15] := 'Buffer';
	bNtSettingsLoadDone : BOOL := TRUE;
END_VAR
(**)
(*Local*)
VAR
	bRstErr : BOOL;
	udiRstErrOld : UDINT;
	bInitDone : BOOL;
	bInitialDone : BOOL;
	bUpdateSensor : BOOL;
	bBffrSetMty : BOOL;
	bBffrSetFull : BOOL;
	bUpdtDisplay : BOOL;
	usiStep : USINT;
	diCurrSlt : DINT;
	diExpectedSlt : DINT;
	bSetFull : BOOL;
	bSetMty : BOOL;
	bCoolFanRun : BOOL;
	tyBffrParameter : tyBffrParam;
	fbDirCreate1 : fbDirCreate;
	fbDirCreate2 : fbDirCreate;
	fbFileRead1 : fbFileFullRead;
	fbFileWrite1 : fbFileFullWrite;
	fbCoolFanOffDlyTm : TON;
	fbCoolFanOffChkTm : TON := (PT:=T#500ms);
	fbMagAbsentTm : TON := (PT:=T#5s);
	fbMagPresentTm : TON := (PT:=T#8s);
	eStatOld : eBufferAction := BufferActIdle;
	bMESTrigSetFull : BOOL;
	udiModuleNum : UDINT := 2001;
END_VAR
```

#### Act_InputConfig.st - not listed in the package file held
```iecst
(** 2019-04-26 **)
ACTION Act_InputConfig:

	(* Always Change If Project Change *)

	//Pass Data To Link
	tylocalBuffer.In.bLinkPresentSen1 := g_tyDInput.bMagPresentSen3;
	tylocalBuffer.In.bLinkPresentSen2 := g_tyDInput.bMagConvEntSen3;
	tylocalBuffer.In.diLinkSltToSltDist ACCESS p_MagRcpCurrRcpSltToSlt;
	tylocalBuffer.In.bLinkMcParamProdSelTopToBtm ACCESS p_ProdRcpCurrRcp2TopToBtm;
	tylocalBuffer.In.bLinkOpsTravLifULExitBrd ACCESS p_OpsTravLifULExitBrd;

	//Pass Data To Internal Use
	tylocalBuffer.In.udiRstErr := g_tyRstErr.bReset;
	tylocalBuffer.In.sFileName := g_tyNtParamCurr.sBffr3FileNm;
	tylocalBuffer.In.bManual := g_tyUIOut.bManualMod;
	tylocalBuffer.In.dtCurrDT := g_tyTime.dtCurrDT;

	tylocalBuffer.In.diBffrTtlSlt ACCESS p_MagRcpCurrRcpTtlSlt;
	tylocalBuffer.In.diLifterBtmPosInUM ACCESS p_MagRcpCurrRcpMag3Slt1Pos;
	tylocalBuffer.In.diLifterCurrPosInUM := g_tyLifterBtm.diActualPos;
	tylocalBuffer.In.bGdBrdIn  := g_tyPshrConv.bGdBrd;
	tylocalBuffer.In.bNxtLoadSeq := g_tyNtParamCurr.bBffr3NxtLoadSeq;
	tylocalBuffer.In.sCurrRcpNm ACCESS p_ProdRcpCurrRcp2Nm;
	tylocalBuffer.In.sProgNm := g_tyNtParamCurr.sBffr3ProgNm;
	tylocalBuffer.In.bNtParamAutoRcpPrep := g_tyNtParamCurr.bAutoRcpPrep ;
	tylocalBuffer.In.bMcParamAutoRcpDis  := g_tyMcParamCurr.bAutoRcpDisable;

	//Siemens Req
	tylocalBuffer.In.bOpsMagConvULRlsMagAllw := g_tyOpsMagConvUL3.bRlsMagAllw;
	tylocalBuffer.In.eNtParamCustomerReq := g_tyNtParamCurr.eCustomerReq;
	tylocalBuffer.In.tyResponseFromMES :=  g_tyAGV.tyTagFromMesMagCov3;

	IF g_tyStartUp.bRun = TRUE THEN
		tylocalBuffer.In.eAct := g_tyStartUp.eBuffer3Act;
	ELSE
		IF tylocalBuffer.Out.eStatus = Idle THEN
			IF g_tyNtParamCurr.bProjLifterMagPlatform = FALSE THEN
				IF g_tyOpsMagConvUL3.eBufferAct <> BufferActIdle THEN
					tylocalBuffer.In.eAct := g_tyOpsMagConvUL3.eBufferAct;
				ELSIF g_tyUIOut.eBuffer3Act <> BufferActIdle THEN
					tylocalBuffer.In.eAct := g_tyUIOut.eBuffer3Act;
				ELSE
					tylocalBuffer.In.eAct := eAct;
				END_IF
			ELSE
				IF g_tyOpsLifMagULBufferAct3.eBufferAct <> BufferActIdle THEN
					tylocalBuffer.In.eAct := g_tyOpsLifMagULBufferAct3.eBufferAct;
				ELSE
					tylocalBuffer.In.eAct := g_tyUIOut.eBuffer3Act;
				END_IF
			END_IF
		END_IF
	END_IF
	(* Always Change If Project Change *)

END_ACTION
```

#### Act_OutputConfig.st - not listed in the package file held
```iecst
(** 2019-06-07 **)
ACTION Act_OutputConfig:

	g_tyBuffer3 := tylocalBuffer.Out;

END_ACTION
```

### Program Logical/Buffer/BufferMagA (IEC) - 1.00.0 - 

#### InputRef.var
```iecst
(*2019-01-30*)
(**)
(*General*)
VAR
	p_bPrep : REFERENCE TO BOOL;
	p_bEn : REFERENCE TO BOOL;
	p_bDis : REFERENCE TO BOOL;
END_VAR
(**)
(*Configuration*)
VAR
	p_eNtParamMag : REFERENCE TO eULMag;
	p_usiMcParamProdSelMcMod : REFERENCE TO USINT;
END_VAR
(**)
VAR
	p_bOpsStatusRun : REFERENCE TO BOOL;
END_VAR
(**)
VAR
	p_bBufferMagPresent1 : REFERENCE TO BOOL;
	p_bBufferMagPresent2 : REFERENCE TO BOOL;
	p_bBufferMagPresent3 : REFERENCE TO BOOL;
	p_bDIMagPresentSen1 : REFERENCE TO BOOL;
	p_bDIMagPresentSen2 : REFERENCE TO BOOL;
	p_bDIMagPresentSen3 : REFERENCE TO BOOL;
END_VAR
(**)
VAR
	p_tyBufferStat1 : REFERENCE TO tyBffrStat;
	p_tyBufferStat2 : REFERENCE TO tyBffrStat;
	p_tyBufferStat3 : REFERENCE TO tyBffrStat;
END_VAR
(*AutoRcp*)
VAR
	p_bNtParamAutoRcpPrep : REFERENCE TO BOOL;
	p_bMcParamAutoRcpDis : REFERENCE TO BOOL;
	p_eNtParamAutoRcpPrecededBy : REFERENCE TO eAutoRcpPreceded;
END_VAR
```

#### Local.var
```iecst
(*2019-01-30*)
(**)
(*Local Action, State & Status*)
(**)
(*Local Alarm*)
(**)
(*Local Output*)
VAR
	diBffrMtySlt : DINT;
END_VAR
(**)
(*Local Input*)
VAR
	bPrep : BOOL := TRUE;
	bEn : BOOL := TRUE;
	bDis : BOOL := FALSE;
	eNtParamMag : eULMag;
	usiMcParamProdSelMcMod : USINT;
	bOpsStatusRun : BOOL;
	bBufferMagPresent1 : BOOL;
	bBufferMagPresent2 : BOOL;
	bBufferMagPresent3 : BOOL;
	tyBufferStat1 : tyBffrStat;
	tyBufferStat2 : tyBffrStat;
	tyBufferStat3 : tyBffrStat;
END_VAR
(**)
(*Local*)
VAR
	bInitDone : BOOL;
	diBffrMtySlt1 : DINT;
	diBffrMtySlt2 : DINT;
	diBffrMtySlt3 : DINT;
END_VAR
```

#### Act_Background.st
```iecst
(** 2019-01-30 **)
ACTION Act_Background:

	(*Lane A - Buffer Empty Slot Algorithm*)

	IF p_bOpsStatusRun = TRUE THEN

		IF p_bBufferMagPresent1 = TRUE AND p_bDIMagPresentSen1 THEN
			diBffrMtySlt1	:= p_tyBufferStat1.diTtlBrdCap - (p_tyBufferStat1.diTtlGdBrd + p_tyBufferStat1.diTtlBadBrd);
		ELSE
			diBffrMtySlt1	:= 0;
		END_IF

		IF p_bBufferMagPresent2 = TRUE AND p_bDIMagPresentSen2 THEN
			diBffrMtySlt2	:= p_tyBufferStat2.diTtlBrdCap - (p_tyBufferStat2.diTtlGdBrd + p_tyBufferStat2.diTtlBadBrd);
		ELSE
			diBffrMtySlt2	:= 0;
		END_IF

		IF p_bBufferMagPresent3 = TRUE AND p_bDIMagPresentSen3 THEN
			diBffrMtySlt3	:= p_tyBufferStat3.diTtlBrdCap - (p_tyBufferStat3.diTtlGdBrd + p_tyBufferStat3.diTtlBadBrd);
		ELSE
			diBffrMtySlt3	:= 0;
		END_IF

		CASE p_eNtParamMag OF
			ULMagDual:

				CASE p_usiMcParamProdSelMcMod OF
					ULModUnloadFrontLnA:

						diBffrMtySlt	:= diBffrMtySlt1 + diBffrMtySlt2;

					ULModRejFrontLnA, ULModRejFrontLnARev, ULModRejDualLnA, ULModRejDualLnB:

						IF diBffrMtySlt2 < diBffrMtySlt1 THEN
							diBffrMtySlt	:= diBffrMtySlt2;
						ELSE
							diBffrMtySlt	:= diBffrMtySlt1;
						END_IF

					ULModUnloadDualLnAB:

						diBffrMtySlt	:= diBffrMtySlt1;

				END_CASE

			ULMagTriple:

				CASE p_usiMcParamProdSelMcMod OF
					ULModUnloadFrontLnA:

						diBffrMtySlt	:= diBffrMtySlt1 + diBffrMtySlt2 + diBffrMtySlt3;

					ULModRejFrontLnA, ULModRejDualLnA:

						IF diBffrMtySlt3 < (diBffrMtySlt1 + diBffrMtySlt2) THEN
							diBffrMtySlt	:= diBffrMtySlt3;
						ELSE
							diBffrMtySlt	:= diBffrMtySlt1 + diBffrMtySlt2;
						END_IF

					ULModRejFrontLnARev, ULModRejDualLnB:

						IF diBffrMtySlt1 < (diBffrMtySlt2 + diBffrMtySlt3) THEN
							diBffrMtySlt	:= diBffrMtySlt1;
						ELSE
							diBffrMtySlt	:= diBffrMtySlt2 + diBffrMtySlt3;
						END_IF

					ULModUnloadDualLnAB:

						diBffrMtySlt	:= diBffrMtySlt1 + diBffrMtySlt2 + diBffrMtySlt3;

				END_CASE

		END_CASE

	END_IF

END_ACTION
```

#### Act_InitGlobal.st
```iecst
(** 2019-01-30 **)
ACTION Act_InitGlobal:

	(* Always Change If Project Change *)

	//Pass Data To Link

	//Pass Data To Internal Use
	p_eNtParamMag ACCESS p_NtParamProjMag;
	p_usiMcParamProdSelMcMod ACCESS p_ProdRcpCurrRcp1McMod;
	p_bOpsStatusRun ACCESS p_OpsStatusRun;
	p_bBufferMagPresent1 ACCESS p_Buffer1MagPresent;
	p_bBufferMagPresent2 ACCESS p_Buffer2MagPresent;
	p_bBufferMagPresent3 ACCESS p_Buffer3MagPresent;
	p_bDIMagPresentSen1 ACCESS p_DIMagPresentSen1;
	p_bDIMagPresentSen2 ACCESS p_DIMagPresentSen2;
	p_bDIMagPresentSen3 ACCESS p_DIMagPresentSen3;

	p_tyBufferStat1 ACCESS p_Buffer1BffrStat;
	p_tyBufferStat2 ACCESS p_Buffer2BffrStat;
	p_tyBufferStat3 ACCESS p_Buffer3BffrStat;

	p_bNtParamAutoRcpPrep ACCESS p_NtParamAutoRcpPrep;
	p_bMcParamAutoRcpDis  ACCESS p_McParamAutoRcpDisable;
	(* Always Change If Project Change *)
	p_eNtParamAutoRcpPrecededBy ACCESS p_NtParamAutoRcpPrecededBy;
END_ACTION
```

#### Act_Initial.st
```iecst
(** 2019-01-30 **)
ACTION Act_Initial:

	//Initial

END_ACTION
```

#### Act_InitLocal.st
```iecst
(** 2019-01-30 **)
ACTION Act_InitLocal:

	//Input Reference Link To Local Variable
	p_bPrep ACCESS ADR(bPrep);
	p_bEn ACCESS ADR(bEn);
	p_bDis ACCESS ADR(bDis);
	p_eNtParamMag ACCESS ADR(eNtParamMag);
	p_usiMcParamProdSelMcMod ACCESS ADR(usiMcParamProdSelMcMod);
	p_bOpsStatusRun ACCESS ADR(bOpsStatusRun);
	p_bBufferMagPresent1 ACCESS ADR(bBufferMagPresent1);
	p_bBufferMagPresent2 ACCESS ADR(bBufferMagPresent2);
	p_bBufferMagPresent3 ACCESS ADR(bBufferMagPresent3);
	p_tyBufferStat1 ACCESS ADR(tyBufferStat1);
	p_tyBufferStat2 ACCESS ADR(tyBufferStat2);
	p_tyBufferStat3 ACCESS ADR(tyBufferStat3);

END_ACTION
```

#### Act_InputConfig.st
```iecst
(** 2019-01-30 **)
ACTION Act_InputConfig:

	(* Always Change If Project Change *)

	//Pass Data To Link

	//Pass Data To Internal Use
	tylocalBufferMag.In.eNtParamMag := g_tyNtParamCurr.eProjMag;
	tylocalBufferMag.In.usiProRcpProdSelMcMod ACCESS p_ProdRcpCurrRcp1McMod;
	tylocalBufferMag.In.bOpsStatusRun := g_tyOps.bStatusRun;
	tylocalBufferMag.In.bBufferMagPresent1 := g_tyBuffer1.bMagPresent;
	tylocalBufferMag.In.bBufferMagPresent2 := g_tyBuffer2.bMagPresent;
	tylocalBufferMag.In.bBufferMagPresent3 := g_tyBuffer3.bMagPresent;
	tylocalBufferMag.In.bDIMagPresentSen1 := g_tyDInput.bMagPresentSen1;
	tylocalBufferMag.In.bDIMagPresentSen2 := g_tyDInput.bMagPresentSen2;
	tylocalBufferMag.In.bDIMagPresentSen3 := g_tyDInput.bMagPresentSen3;

	tylocalBufferMag.In.tyBufferStat1 := g_tyBuffer1.tyBufferStat;
	tylocalBufferMag.In.tyBufferStat2 := g_tyBuffer2.tyBufferStat;
	tylocalBufferMag.In.tyBufferStat3 := g_tyBuffer3.tyBufferStat;

	tylocalBufferMag.In.bNtParamAutoRcpPrep := g_tyNtParamCurr.bAutoRcpPrep;
	tylocalBufferMag.In.bMcParamAutoRcpDis  := g_tyMcParamCurr.bAutoRcpDisable;
	(* Always Change If Project Change *)

END_ACTION
```

#### Act_Link.st
```iecst
(** 2019-01-30 **)
ACTION Act_Link:

	IF p_bNtParamAutoRcpPrep AND NOT(p_bMcParamAutoRcpDis) AND p_eNtParamAutoRcpPrecededBy = PrecededBySelf THEN //AutoRcp Ignored Follower
		p_usiMcParamProdSelMcMod ACCESS p_ProdRcpCurrRcp0McMod;
	ELSE
		p_usiMcParamProdSelMcMod ACCESS p_ProdRcpCurrRcp1McMod;
	END_IF

END_ACTION
```

#### Act_Main.st
```iecst
(** 2019-01-30 **)
ACTION Act_Main:

		(*Lane A - Buffer Empty Slot Algorithm*)

	IF tylocalBufferMag.In.bOpsStatusRun = TRUE THEN

		IF tylocalBufferMag.In.bBufferMagPresent1 = TRUE AND tylocalBufferMag.In.bDIMagPresentSen1 THEN
			diBffrMtySlt1	:= tylocalBufferMag.In.tyBufferStat1.diTtlBrdCap - (tylocalBufferMag.In.tyBufferStat1.diTtlGdBrd + tylocalBufferMag.In.tyBufferStat1.diTtlBadBrd);
		ELSE
			diBffrMtySlt1	:= 0;
		END_IF

		IF tylocalBufferMag.In.bBufferMagPresent2 = TRUE AND tylocalBufferMag.In.bDIMagPresentSen2 THEN
			diBffrMtySlt2	:= tylocalBufferMag.In.tyBufferStat2.diTtlBrdCap - (tylocalBufferMag.In.tyBufferStat2.diTtlGdBrd + tylocalBufferMag.In.tyBufferStat2.diTtlBadBrd);
		ELSE
			diBffrMtySlt2	:= 0;
		END_IF

		IF tylocalBufferMag.In.bBufferMagPresent3 = TRUE AND tylocalBufferMag.In.bDIMagPresentSen3 THEN
			diBffrMtySlt3	:= tylocalBufferMag.In.tyBufferStat3.diTtlBrdCap - (tylocalBufferMag.In.tyBufferStat3.diTtlGdBrd + tylocalBufferMag.In.tyBufferStat3.diTtlBadBrd);
		ELSE
			diBffrMtySlt3	:= 0;
		END_IF

		CASE tylocalBufferMag.In.eNtParamMag OF
			ULMagDual:

				CASE tylocalBufferMag.In.usiProRcpProdSelMcMod OF
					ULModUnloadFrontLnA:

						tylocalBufferMag.Out.diBffrMtySlt	:= diBffrMtySlt1 + diBffrMtySlt2;

					ULModRejFrontLnA, ULModRejFrontLnARev, ULModRejDualLnA, ULModRejDualLnB:

						IF diBffrMtySlt2 < diBffrMtySlt1 THEN
							tylocalBufferMag.Out.diBffrMtySlt	:= diBffrMtySlt2;
						ELSE
							tylocalBufferMag.Out.diBffrMtySlt	:= diBffrMtySlt1;
						END_IF

					ULModUnloadDualLnAB:

						tylocalBufferMag.Out.diBffrMtySlt	:= diBffrMtySlt1;

				END_CASE

			ULMagTriple:

				CASE tylocalBufferMag.In.usiProRcpProdSelMcMod OF
					ULModUnloadFrontLnA:

						tylocalBufferMag.Out.diBffrMtySlt	:= diBffrMtySlt1 + diBffrMtySlt2 + diBffrMtySlt3;

					ULModRejFrontLnA, ULModRejDualLnA:

						IF diBffrMtySlt3 < (diBffrMtySlt1 + diBffrMtySlt2) THEN
							tylocalBufferMag.Out.diBffrMtySlt	:= diBffrMtySlt3;
						ELSE
							tylocalBufferMag.Out.diBffrMtySlt	:= diBffrMtySlt1 + diBffrMtySlt2;
						END_IF

					ULModRejFrontLnARev, ULModRejDualLnB:

						IF diBffrMtySlt1 < (diBffrMtySlt2 + diBffrMtySlt3) THEN
							tylocalBufferMag.Out.diBffrMtySlt	:= diBffrMtySlt1;
						ELSE
							tylocalBufferMag.Out.diBffrMtySlt	:= diBffrMtySlt2 + diBffrMtySlt3;
						END_IF

					ULModUnloadDualLnAB:

						tylocalBufferMag.Out.diBffrMtySlt	:= diBffrMtySlt1 + diBffrMtySlt2 + diBffrMtySlt3;

				END_CASE

		END_CASE

	END_IF

END_ACTION
```

#### Act_OutputConfig.st
```iecst
(** 2019-01-30 **)
ACTION Act_OutputConfig:

	g_tyBufferMagA := tylocalBufferMag.Out;

END_ACTION
```

#### Cyclic.st
```iecst
(** 2019-01-30 **)
PROGRAM _CYCLIC

	IF bInitDone = FALSE THEN
		bInitDone	:= TRUE;
		Act_Initial;

	ELSE
		Act_InputConfig;
		IF (tylocalBufferMagA.In.bPrep = TRUE) AND (tylocalBufferMagA.In.bEn = TRUE) AND (tylocalBufferMagA.In.bDis = FALSE) THEN
			Act_Link;
			Act_Main;
		ELSE
			Act_Main_Disable;
		END_IF
		Act_OutputConfig;
	END_IF

END_PROGRAM
```

#### Init.st
```iecst
(** 2019-01-30 **)
PROGRAM _INIT

	(* Always Change If Project Change *)

	//Pass Address To Global Address For External Use
	//Action, State & Status

	//Alarm

	//Output
	p_BufferMagABffrMtySlt	:= ADR(diBffrMtySlt);

	(* Always Change If Project Change *)

END_PROGRAM
```

### Program Logical/Buffer/BufferMagB (IEC, version 1.00.0) - 1.00.0 - 

#### Act_InputConfig.st - Change By Project
```iecst
(** 2019-01-30 **)
ACTION Act_InputConfig:

	(* Always Change If Project Change *)

	//Pass Data To Link

	//Pass Data To Internal Use
	tylocalBufferMag.In.eNtParamMag := g_tyNtParamCurr.eProjMag;
	tylocalBufferMag.In.usiProRcpProdSelMcMod ACCESS p_ProdRcpCurrRcp1McMod;
	tylocalBufferMag.In.bOpsStatusRun := g_tyOps.bStatusRun;
	tylocalBufferMag.In.bBufferMagPresent1 := g_tyBuffer1.bMagPresent;
	tylocalBufferMag.In.bBufferMagPresent2 := g_tyBuffer2.bMagPresent;
	tylocalBufferMag.In.bBufferMagPresent3 := g_tyBuffer3.bMagPresent;
	tylocalBufferMag.In.bDIMagPresentSen1 := g_tyDInput.bMagPresentSen1;
	tylocalBufferMag.In.bDIMagPresentSen2 := g_tyDInput.bMagPresentSen2;
	tylocalBufferMag.In.bDIMagPresentSen3 := g_tyDInput.bMagPresentSen3;

	tylocalBufferMag.In.tyBufferStat1 := g_tyBuffer1.BffrStat;
	tylocalBufferMag.In.tyBufferStat2 := g_tyBuffer2.BffrStat;
	tylocalBufferMag.In.tyBufferStat3 := g_tyBuffer3.BffrStat;

	tylocalBufferMag.In.bNtParamAutoRcpPrep := g_tyNtParamCurr.bAutoRcpPrep;
	tylocalBufferMag.In.bMcParamAutoRcpDis  := g_tyMcParamCurr.bAutoRcpDisable;
	(* Always Change If Project Change *)

END_ACTION
```

#### Act_OutputConfig.st - Change By Project
```iecst
(** 2019-01-30 **)
ACTION Act_OutputConfig:

	g_tyBufferMagB := tylocalBufferMag.Out;

END_ACTION
```

#### Act_Link.st - Change By Project
```iecst
(** 2019-01-30 **)
ACTION Act_Link:

	IF tylocalBufferMag.In.bNtParamAutoRcpPrep AND NOT(tylocalBufferMag.In.bMcParamAutoRcpDis) THEN //AutoRcp Ignored Follower
		tylocalBufferMag.In.usiProRcpProdSelMcMod ACCESS p_ProdRcpCurrRcp0McMod;
	ELSE
		tylocalBufferMag.In.usiProRcpProdSelMcMod ACCESS p_ProdRcpCurrRcp1McMod;
	END_IF

END_ACTION
```

#### Act_Main.st - Do Not Change!!!
```iecst
(** 2019-01-30 **)
ACTION Act_Main:

		(*Lane B - Buffer Empty Slot Algorithm*)

	IF tylocalBufferMag.In.bOpsStatusRun = TRUE THEN

		IF tylocalBufferMag.In.bBufferMagPresent1 = TRUE AND tylocalBufferMag.In.bDIMagPresentSen1 THEN
			diBffrMtySlt1	:= tylocalBufferMag.In.tyBufferStat1.diTtlBrdCap - (tylocalBufferMag.In.tyBufferStat1.diTtlGdBrd + tylocalBufferMag.In.tyBufferStat1.diTtlBadBrd);
		ELSE
			diBffrMtySlt1	:= 0;
		END_IF

		IF tylocalBufferMag.In.bBufferMagPresent2 = TRUE AND tylocalBufferMag.In.bDIMagPresentSen2 THEN
			diBffrMtySlt2	:= tylocalBufferMag.In.tyBufferStat2.diTtlBrdCap - (tylocalBufferMag.In.tyBufferStat2.diTtlGdBrd + tylocalBufferMag.In.tyBufferStat2.diTtlBadBrd);
		ELSE
			diBffrMtySlt2	:= 0;
		END_IF

		IF tylocalBufferMag.In.bBufferMagPresent3 = TRUE AND tylocalBufferMag.In.bDIMagPresentSen3 THEN
			diBffrMtySlt3	:= tylocalBufferMag.In.tyBufferStat3.diTtlBrdCap - (tylocalBufferMag.In.tyBufferStat3.diTtlGdBrd + tylocalBufferMag.In.tyBufferStat3.diTtlBadBrd);
		ELSE
			diBffrMtySlt3	:= 0;
		END_IF

		CASE tylocalBufferMag.In.eNtParamMag OF
			ULMagDual:

				CASE tylocalBufferMag.In.usiMcParamProdSelMcMod OF
					ULModUnloadRearLnB:

						tylocalBufferMag.Out.diBffrMtySlt	:= diBffrMtySlt1 + diBffrMtySlt2;

					ULModRejRearLnB, ULModRejRearLnBRev, ULModRejDualLnA, ULModRejDualLnB:

						IF diBffrMtySlt2 < diBffrMtySlt1 THEN
							tylocalBufferMag.Out.diBffrMtySlt	:= diBffrMtySlt2;
						ELSE
							tylocalBufferMag.Out.diBffrMtySlt	:= diBffrMtySlt1;
						END_IF

					ULModUnloadDualLnAB:

						tylocalBufferMag.Out.diBffrMtySlt	:= diBffrMtySlt2;

				END_CASE

			ULMagTriple:

				CASE tylocalBufferMag.In.usiMcParamProdSelMcMod OF
					ULModUnloadRearLnB:

						tylocalBufferMag.Out.diBffrMtySlt	:= diBffrMtySlt1 + diBffrMtySlt2 + diBffrMtySlt3;

					ULModRejRearLnB, ULModRejDualLnB:

						IF diBffrMtySlt1 < (diBffrMtySlt2 + diBffrMtySlt3) THEN
							tylocalBufferMag.Out.diBffrMtySlt	:= diBffrMtySlt1;
						ELSE
							tylocalBufferMag.Out.diBffrMtySlt	:= diBffrMtySlt2 + diBffrMtySlt3;
						END_IF

					ULModRejRearLnBRev, ULModRejDualLnA:

						IF diBffrMtySlt3 < (diBffrMtySlt1 + diBffrMtySlt2) THEN
							tylocalBufferMag.Out.diBffrMtySlt	:= diBffrMtySlt3;
						ELSE
							tylocalBufferMag.Out.diBffrMtySlt	:= diBffrMtySlt1 + diBffrMtySlt2;
						END_IF

					ULModUnloadDualLnAB:

						tylocalBufferMag.Out.diBffrMtySlt	:= diBffrMtySlt1 + diBffrMtySlt2 + diBffrMtySlt3;

				END_CASE

		END_CASE

	END_IF

END_ACTION
```

#### Act_Main_Disable.st - Do Not Change!!!
```iecst
(** 2019-01-30 **)
ACTION Act_Main_Disable:

	tylocalBufferMag.Out.diBffrMtySlt	:= 0;

END_ACTION
```

#### Local.var - Do Not Change!!!
```iecst
(*2019-01-30*)
(**)
(*Local Action, State & Status*)
(**)
(*Local Alarm*)
VAR
	tylocalBufferMag : tyBufferMag;
END_VAR
(**)
(*Local*)
VAR
	bInitDone : BOOL;
	diBffrMtySlt1 : DINT;
	diBffrMtySlt2 : DINT;
	diBffrMtySlt3 : DINT;
END_VAR
```

#### InputRef.var - not listed in the package file held
```iecst
(*2019-01-30*)
(**)
(*General*)
VAR
	p_bPrep : REFERENCE TO BOOL;
	p_bEn : REFERENCE TO BOOL;
	p_bDis : REFERENCE TO BOOL;
END_VAR
(**)
(*Configuration*)
VAR
	p_eNtParamMag : REFERENCE TO eULMag;
	p_usiMcParamProdSelMcMod : REFERENCE TO USINT;
END_VAR
(**)
VAR
	p_bOpsStatusRun : REFERENCE TO BOOL;
END_VAR
(**)
VAR
	p_bBufferMagPresent1 : REFERENCE TO BOOL;
	p_bBufferMagPresent2 : REFERENCE TO BOOL;
	p_bBufferMagPresent3 : REFERENCE TO BOOL;
	p_bDIMagPresentSen1 : REFERENCE TO BOOL;
	p_bDIMagPresentSen2 : REFERENCE TO BOOL;
	p_bDIMagPresentSen3 : REFERENCE TO BOOL;
END_VAR
(**)
VAR
	p_tyBufferStat1 : REFERENCE TO tyBffrStat;
	p_tyBufferStat2 : REFERENCE TO tyBffrStat;
	p_tyBufferStat3 : REFERENCE TO tyBffrStat;
END_VAR
(*AutoRcp*)
VAR
	p_bNtParamAutoRcpPrep : REFERENCE TO BOOL;
	p_bMcParamAutoRcpDis : REFERENCE TO BOOL;
END_VAR
```

#### Act_Action.st - not listed in the package file held
```iecst
(** 2019-01-30 **)
ACTION Act_Action:

	//Set eAct

END_ACTION
```

#### Act_Background.st - not listed in the package file held
```iecst
(** 2019-01-30 **)
ACTION Act_Background:

	(*Lane B - Buffer Empty Slot Algorithm*)

	IF p_bOpsStatusRun = TRUE THEN

		IF p_bBufferMagPresent1 = TRUE AND p_bDIMagPresentSen1 THEN
			diBffrMtySlt1	:= p_tyBufferStat1.diTtlBrdCap - (p_tyBufferStat1.diTtlGdBrd + p_tyBufferStat1.diTtlBadBrd);
		ELSE
			diBffrMtySlt1	:= 0;
		END_IF

		IF p_bBufferMagPresent2 = TRUE AND p_bDIMagPresentSen2 THEN
			diBffrMtySlt2	:= p_tyBufferStat2.diTtlBrdCap - (p_tyBufferStat2.diTtlGdBrd + p_tyBufferStat2.diTtlBadBrd);
		ELSE
			diBffrMtySlt2	:= 0;
		END_IF

		IF p_bBufferMagPresent3 = TRUE AND p_bDIMagPresentSen3 THEN
			diBffrMtySlt3	:= p_tyBufferStat3.diTtlBrdCap - (p_tyBufferStat3.diTtlGdBrd + p_tyBufferStat3.diTtlBadBrd);
		ELSE
			diBffrMtySlt3	:= 0;
		END_IF

		CASE p_eNtParamMag OF
			ULMagDual:

				CASE p_usiMcParamProdSelMcMod OF
					ULModUnloadRearLnB:

						diBffrMtySlt	:= diBffrMtySlt1 + diBffrMtySlt2;

					ULModRejRearLnB, ULModRejRearLnBRev, ULModRejDualLnA, ULModRejDualLnB:

						IF diBffrMtySlt2 < diBffrMtySlt1 THEN
							diBffrMtySlt	:= diBffrMtySlt2;
						ELSE
							diBffrMtySlt	:= diBffrMtySlt1;
						END_IF

					ULModUnloadDualLnAB:

						diBffrMtySlt	:= diBffrMtySlt2;

				END_CASE

			ULMagTriple:

				CASE p_usiMcParamProdSelMcMod OF
					ULModUnloadRearLnB:

						diBffrMtySlt	:= diBffrMtySlt1 + diBffrMtySlt2 + diBffrMtySlt3;

					ULModRejRearLnB, ULModRejDualLnB:

						IF diBffrMtySlt1 < (diBffrMtySlt2 + diBffrMtySlt3) THEN
							diBffrMtySlt	:= diBffrMtySlt1;
						ELSE
							diBffrMtySlt	:= diBffrMtySlt2 + diBffrMtySlt3;
						END_IF

					ULModRejRearLnBRev, ULModRejDualLnA:

						IF diBffrMtySlt3 < (diBffrMtySlt1 + diBffrMtySlt2) THEN
							diBffrMtySlt	:= diBffrMtySlt3;
						ELSE
							diBffrMtySlt	:= diBffrMtySlt1 + diBffrMtySlt2;
						END_IF

					ULModUnloadDualLnAB:

						diBffrMtySlt	:= diBffrMtySlt1 + diBffrMtySlt2 + diBffrMtySlt3;

				END_CASE

		END_CASE

	END_IF

END_ACTION
```

#### Act_InitGlobal.st - not listed in the package file held
```iecst
(** 2019-01-30 **)
ACTION Act_InitGlobal:

	(* Always Change If Project Change *)

	//Pass Data To Link

	//Pass Data To Internal Use
	p_eNtParamMag ACCESS p_NtParamProjMag;
	//p_usiMcParamProdSelMcMod ACCESS p_ProdRcpCurrRcp1McMod;
	p_bOpsStatusRun ACCESS p_OpsStatusRun;
	p_bBufferMagPresent1 ACCESS p_Buffer1MagPresent;
	p_bBufferMagPresent2 ACCESS p_Buffer2MagPresent;
	p_bBufferMagPresent3 ACCESS p_Buffer3MagPresent;
	p_bDIMagPresentSen1 ACCESS p_DIMagPresentSen1;
	p_bDIMagPresentSen2 ACCESS p_DIMagPresentSen2;
	p_bDIMagPresentSen3 ACCESS p_DIMagPresentSen3;
	p_tyBufferStat1 ACCESS p_Buffer1BffrStat;
	p_tyBufferStat2 ACCESS p_Buffer2BffrStat;
	p_tyBufferStat3 ACCESS p_Buffer3BffrStat;

	p_bNtParamAutoRcpPrep ACCESS p_NtParamAutoRcpPrep;
	p_bMcParamAutoRcpDis  ACCESS p_McParamAutoRcpDisable;
	(* Always Change If Project Change *)
	p_eNtParamAutoRcpPrecededBy ACCESS p_NtParamAutoRcpPrecededBy;
END_ACTION
```

#### Act_LinkEn.st - not listed in the package file held
```iecst
(** 2019-01-30 **)
ACTION Act_LinkEn:

	//Link bPrep, bEn & bDis

END_ACTION
```

#### Init.st - not listed in the package file held
```iecst
(** 2019-01-30 **)
PROGRAM _INIT

	(* Always Change If Project Change *)

	//Pass Address To Global Address For External Use
	//Action, State & Status

	//Alarm

	//Output
	p_BufferMagBBffrMtySlt	:= ADR(diBffrMtySlt);

	(* Always Change If Project Change *)

END_PROGRAM
```
